CASE eCommand OF
	MC_NoCmd :
		CASE sCurrentState.eStatus OF
			MS_Init :
				IF bEnable THEN
					CASE sCurrentState.eStep OF
						SP_InitStp1 : (* Init all synchros *)
							bBarrelNeedScan := FALSE;
							bArea1StickWarning := FALSE;
							bArea2StickWarning := FALSE;
							bArea3StickWarning := FALSE;
							bArea4StickWarning := FALSE;
							FOR i:=1 TO iMaxSection DO
								FOR j:=1 TO iMaxPosition DO
									abStickPresent[1,i,j]:= FALSE;
									abStickPresent[2,i,j]:= FALSE;
								END_FOR
							END_FOR
							sCurrentState.eStep := SP_InitStp2;
						SP_InitStp2 : (* Lower jacks *)
							bMoveJackUp := FALSE;
							sCurrentState.eStep := SP_InitStp3;
						SP_InitStp3 : (* Check if jacks are down *)
							IF bJackIsDown THEN
								sCurrentState.eStep := SP_InitStp4;
							END_IF
						SP_InitStp4 : (* Lower index *)
							bIndexTable := FALSE;
							sCurrentState.eStep := SP_InitStp5;
						SP_InitStp5 : (* Check if index are down *)
							IF bJackIsDown AND bTableNotIndexed THEN
								sCurrentState.eStep := SP_InitStp6;
							END_IF
						SP_InitStp6 : (* Init barrel axis if modules are safe*)
							eMoveBarrelAxisCommand := AC_Init;
							sCurrentState.eStep := SP_InitStp7;
						SP_InitStp7 : (* Wait init barrel is done*)
							IF TBarrelAxis.eCurrentState = AS_InPosition THEN
								IF bUseNewBarrelFunction THEN
									sCurrentState.eStep := SP_InitStp30;
								ELSE
									sCurrentState.eStep := SP_InitStp10;
								END_IF
							END_IF
						SP_InitStp10 : (* Mono section to use *)
							iIndexPosition := 1;
							IF NOT bSection1IsUsed AND NOT bSection2IsUsed THEN (* no section used *)
								iIndexSection := 1;
								sCurrentState.eStep := SP_InitStp17;
							ELSIF NOT bSection1IsUsed THEN (* section 1 not used *)
								iIndexSection := iStickUsedSection2 + 1;
								iScanPearling:= 2;
								bStickFound := FALSE;
								sCurrentState.eStep := SP_InitStp11;
							ELSE
								iIndexSection := iStickUsedSection1 + 1;
								iScanPearling:= 1;
								bStickFound := FALSE;
								sCurrentState.eStep := SP_InitStp11;
							END_IF
						SP_InitStp11 : (* Turn the barrel to go to the check stick*)
							lrBarrelTargetPos := alrIndexSectionPosition[iIndexSection, iIndexPosition] + lrBarrelCheckPos - alrIndexSectionPosition[1, 1];
							eMoveBarrelAxisCommand := AC_MoveAtAbsPos;
							bStartTimer := FALSE;
							sCurrentState.eStep := SP_InitStp13;
						SP_InitStp13 : (* Wait until position is reached to start the timer *)
							IF (TBarrelAxis.eCurrentState = AS_InPosition) THEN
								bStartTimer := TRUE;
								sCurrentState.eStep := SP_InitStp15;
							END_IF
						SP_InitStp15: (* Wait until the end of timer to detect if the stick is here *)
							IF TBarrelDetectionTimer.Q THEN
								bStartTimer := FALSE;
								abStickPresent[iScanPearling,iIndexSection, iIndexPosition] := bStickPresent;
								IF (bStickPresent) THEN bStickFound := TRUE; END_IF
								iIndexPosition := iIndexPosition + 1;
								IF (iIndexPosition > iMaxPosition) THEN
									CASE iIndexSection OF
										1 :
											bArea1StickWarning := NOT bStickFound;
										2 :
											bArea2StickWarning := NOT bStickFound;
										3 :
											bArea3StickWarning := NOT bStickFound;
										4 :
											bArea4StickWarning := NOT bStickFound;
									END_CASE
									bStickFound := FALSE;
									iIndexPosition := 1;
									iScanPearling:=iScanPearling + 1;
									IF (iScanPearling > 2)  OR (iStickUsedSection1 = iStickUsedSection2) OR NOT bSection2IsUsed THEN
										IF NOT bSection1IsUsed THEN
											iIndexSection := iStickUsedSection2 + 1;
										ELSE
											iIndexSection := iStickUsedSection1 + 1;
										END_IF
										sCurrentState.eStep := SP_InitStp17;
									ELSE
										iIndexSection:= iStickUsedSection2 + 1;
										sCurrentState.eStep := SP_InitStp11;
									END_IF
								ELSE
									sCurrentState.eStep := SP_InitStp11;
								END_IF
							END_IF
						SP_InitStp17 : (* Move to taken,section used 1, 1 *)
							lrBarrelTargetPos := alrIndexSectionPosition[iIndexSection, iIndexPosition] + lrBarrelTakenPos - alrIndexSectionPosition[1, 1];
							eMoveBarrelAxisCommand := AC_MoveAtAbsPos;
							sCurrentState.eStep := SP_InitStp19;
						SP_InitStp19 : (* Wait until position is reached  *)
							IF (TBarrelAxis.eCurrentState = AS_InPosition) THEN
								sCurrentState.eStep := SP_InitStp99;
							END_IF
						SP_InitStp30 : (* Multi section to use *)
							iIndexPosition := 1;
							IF NOT bSection1IsUsed AND NOT bSection2IsUsed THEN (* no section used *)
								iIndexSection := 1;
								sCurrentState.eStep := SP_InitStp37;
							ELSIF NOT bSection1IsUsed THEN (* section 1 not used *)
								yMultiSection2Use := INT_TO_BYTE(iStickUsedSection2);
								iScanPearling:= 2;
								bStickFound := FALSE;
								sCurrentState.eStep := SP_InitStp31;
							ELSE
								yMultiSection2Use := INT_TO_BYTE(iStickUsedSection1);
								iScanPearling:= 1;
								bStickFound := FALSE;
								sCurrentState.eStep := SP_InitStp31;
							END_IF
						SP_InitStp31 :
							iIndexSection := BYTE_TO_INT( yGetActiveSection(yMultiSection2Use));
							IF iIndexSection = 0 THEN
								iIndexSection := 1;
								sCurrentState.eStep := SP_InitStp37;
							ELSE
								sCurrentState.eStep := SP_InitStp32;
							END_IF
						SP_InitStp32 : (* Turn the barrel to go to the check stick*)
							lrBarrelTargetPos := alrIndexSectionPosition[iIndexSection, iIndexPosition] + lrBarrelCheckPos - alrIndexSectionPosition[1, 1];
							eMoveBarrelAxisCommand := AC_MoveAtAbsPos;
							bStartTimer := FALSE;
							sCurrentState.eStep := SP_InitStp33;
						SP_InitStp33 : (* Wait until position is reached to start the timer *)
							IF (TBarrelAxis.eCurrentState = AS_InPosition) THEN
								bStartTimer := TRUE;
								sCurrentState.eStep := SP_InitStp35;
							END_IF
						SP_InitStp35: (* Wait until the end of timer to detect if the stick is here *)
							IF TBarrelDetectionTimer.Q THEN
								bStartTimer := FALSE;
								abStickPresent[iScanPearling,iIndexSection, iIndexPosition] := bStickPresent;
								IF (bStickPresent) THEN bStickFound := TRUE; END_IF
								iIndexPosition := iIndexPosition + 1;
								IF (iIndexPosition > iMaxPosition) THEN
									CASE iIndexSection OF
										1 :
											bArea1StickWarning := NOT bStickFound;
										2 :
											bArea2StickWarning := NOT bStickFound;
										3 :
											bArea3StickWarning := NOT bStickFound;
										4 :
											bArea4StickWarning := NOT bStickFound;
									END_CASE
									bStickFound := FALSE;
									iIndexPosition := 1;
									iIndexSection := BYTE_TO_INT(yGetActiveSection(yMultiSection2Use));
									IF iIndexSection = 0 THEN
										iScanPearling:=iScanPearling + 1;
(*										IF (iScanPearling > 2)  OR (iStickUsedSection1 = iStickUsedSection2) OR NOT bSection2IsUsed THEN*)
										IF (iScanPearling > 2)  OR NOT bSection2IsUsed THEN
											IF NOT bSection1IsUsed THEN
												yMultiSection2Use := INT_TO_BYTE(iStickUsedSection2);
												iIndexSection := BYTE_TO_INT( yGetActiveSection(yMultiSection2Use));
											ELSE
												yMultiSection2Use := INT_TO_BYTE(iStickUsedSection1);
												iIndexSection := BYTE_TO_INT( yGetActiveSection(yMultiSection2Use));
											END_IF
											sCurrentState.eStep := SP_InitStp37;
										ELSE
											yMultiSection2Use := INT_TO_BYTE(iStickUsedSection2);
											sCurrentState.eStep := SP_InitStp31;
										END_IF
									ELSE
										sCurrentState.eStep := SP_InitStp32;
									END_IF
								ELSE
									sCurrentState.eStep := SP_InitStp32;
								END_IF
							END_IF
						SP_InitStp37 : (* Move to taken,section used 1, 1 *)
							lrBarrelTargetPos := alrIndexSectionPosition[iIndexSection, iIndexPosition] + lrBarrelTakenPos - alrIndexSectionPosition[1, 1];
							eMoveBarrelAxisCommand := AC_MoveAtAbsPos;
							sCurrentState.eStep := SP_InitStp39;
						SP_InitStp39 : (* Wait until position is reached  *)
							IF (TBarrelAxis.eCurrentState = AS_InPosition) THEN
								sCurrentState.eStep := SP_InitStp99;
							END_IF
						SP_InitStp99 : (* Leave Init *)
							sCurrentState.eStep := SP_RunStp1;
							sCurrentState.eStatus := MS_Ready;
							sCurrentState.bInitDone := TRUE;
					END_CASE
				ELSE
					sCurrentState.eStatus := MS_Ready;
					sCurrentState.bInitDone := TRUE;
				END_IF
			MS_Running :
				IF bEnable AND  (NOT sCurrentState.bWaitStep) THEN
					CASE sCurrentState.eStep OF
						SP_RunStp1:
							eRunStatus := RS_WaitRequest;
							CASE eRunCommand OF
								RCB_None:
									IF bStopReq  THEN
										sCurrentState.eStatus := MS_Ready;
									ELSIF bPauseReq THEN
										sCurrentState.eStatus := MS_Paused;
									END_IF
								RCB_PrepareStick:
									sCurrentState.eStep := SP_RunStp10;
								RCB_GiveStick:
									sOutStickTake.bHasGiven := FALSE;
									sCurrentState.eStep := SP_RunStp20;
							END_CASE
							IF sCurrentState.eStep<> SP_RunStp1 THEN eRunStatus := RS_ProcessRequest1; END_IF
						SP_RunStp10:(* Prepare Stick *)
							 (* Search Stick *)
							iSearchIndexPosition := 0;
							FOR j:=1 TO 4 DO
								FOR i:=1 TO iMaxPosition DO
									IF abStickPresent[iStickArea,j,i] THEN
										iSearchIndexSection := j;
										iSearchIndexPosition := i;
										EXIT;
									END_IF
								END_FOR
							END_FOR
							IF iSearchIndexPosition = 0 THEN
								bBarrelEmptyError := TRUE;
								sCurrentState.eStep := SP_RunStp1;
							ELSIF iIndexPosition=iSearchIndexPosition AND iIndexSection=iSearchIndexSection AND bTableIndexed THEN
								(* Already prepared *)
								sCurrentState.eStep := SP_RunStp1;
							ELSE
								iIndexPosition := iSearchIndexPosition;
								 iIndexSection := iSearchIndexSection;
								sCurrentState.eStep := SP_RunStp11;
							END_IF
						SP_RunStp11:
							(* Unlock table *)
							bMoveJackUp := FALSE;
							bIndexTable := FALSE;
							sCurrentState.eStep := SP_RunStp12;
						SP_RunStp12: (* Ready to move *)
							IF bJackIsDown AND bTableNotIndexed THEN
								sCurrentState.eStep := SP_RunStp13;
							END_IF
						SP_RunStp13: (* Move to Stick *)
							lrBarrelTargetPos := alrIndexSectionPosition[iIndexSection, iIndexPosition] + lrBarrelTakenPos - alrIndexSectionPosition[1, 1];
							eMoveBarrelAxisCommand := AC_MoveAtAbsPos;
							sCurrentState.eStep := SP_RunStp14;
						SP_RunStp14 : (* Wait until position is reached*)
							IF (TBarrelAxis.eCurrentState = AS_InPosition) THEN
								(* Lock table *)
								bIndexTable := TRUE;
								sCurrentState.eStep := SP_RunStp15;
							END_IF
						SP_RunStp15 :
							IF bTableIndexed THEN
								sCurrentState.eStep := SP_RunStp1;
							END_IF
						SP_RunStp20 : (* Raise the jack when pearling ready*)
							IF NOT bTableIndexed THEN
								bCommandError := TRUE;
							END_IF
							bMoveJackUp := FALSE;
							IF bTableIndexed AND bJackisDown AND sInStickTake.bReadyToTake THEN
								bBarrelNeedScan := TRUE;
								bMoveJackUp := TRUE;
								sCurrentState.eStep := SP_RunStp21;
							END_IF
						SP_RunStp21 : (* Wait for the jack to be up *)
							IF bJackisUp THEN
								sOutStickTake.bHasGiven := TRUE;
								sCurrentState.eStep := SP_RunStp22;
							END_IF
						SP_RunStp22 : (* Wait until the broach has taken the stick *)
							IF sInStickTake.bHasTaken THEN
								sCurrentState.eStep := SP_RunStp23;
							END_IF
						SP_RunStp23 : (* Lower the jack *)
							bMoveJackUp := FALSE;
							sCurrentState.eStep := SP_RunStp24;
						SP_RunStp24 : (* Wait for the jack to go in *)
							IF bJackisDown THEN
								(* Unlock table *)
								bIndexTable := FALSE;
								sCurrentState.eStep := SP_RunStp25;
							END_IF
						SP_RunStp25: (* Check if the stick is still here *)
							IF bTableNotIndexed THEN
								lrBarrelTargetPos := alrIndexSectionPosition[iIndexSection, iIndexPosition] + lrBarrelCheckPos - alrIndexSectionPosition[1, 1];
								eMoveBarrelAxisCommand := AC_MoveAtAbsPos;
								bStartTimer := FALSE;
								sCurrentState.eStep := SP_RunStp26;
							END_IF
						SP_RunStp26 : (* Wait until position is reached to start the timer *)
							IF (TBarrelAxis.eCurrentState = AS_InPosition) THEN
								bStartTimer := TRUE;
								sCurrentState.eStep := SP_RunStp27;
							END_IF
						SP_RunStp27: (* Wait until the end of timer to detect if the stick is still here *)
							IF TBarrelDetectionTimer.Q THEN
								bStartTimer := FALSE;
								abStickPresent[1,iIndexSection, iIndexPosition] := bStickPresent;
								abStickPresent[2,iIndexSection, iIndexPosition] := bStickPresent;
								bBarrelNeedScan := FALSE;
								sOutStickTake.bHasGiven := NOT bStickPresent;
								sCurrentState.eStep := SP_RunStp1;
							END_IF
					END_CASE
				END_IF
			MS_Manual :
				IF NOT bPowerOn THEN
					TManualCmd.TMoveJackUp.Activate := FALSE;
					TManualCmd.TIndexTable.Activate := FALSE;
				END_IF
				TManualCmd.TBarrelAxis.Home.Enable := bJackIsDown AND bTableNotIndexed AND ((TBarrelAxis.eCurrentState = AS_InPosition) OR (TBarrelAxis.eCurrentState = AS_NotHomed)) AND NOT 
bManInterlock;
				TManualCmd.TBarrelAxis.MoveBw.Enable := TBarrelAxis.eCurrentState = AS_InPosition AND bJackIsDown AND bTableNotIndexed AND NOT bManInterlock;
				TManualCmd.TBarrelAxis.MoveFw.Enable := TManualCmd.TBarrelAxis.MoveBw.Enable;
				TManualCmd.TBarrelAxisTakenPos.MoveToTeach.Enable := TManualCmd.TBarrelAxis.MoveBw.Enable;
				TManualCmd.TMoveTaken.TMove1Step.Enable := TManualCmd.TBarrelAxis.MoveBw.Enable;
				TManualCmd.TMoveTaken.TMoveSectionA.Enable := TManualCmd.TBarrelAxis.MoveBw.Enable;
				TManualCmd.TMoveTaken.TMoveSectionB.Enable := TManualCmd.TBarrelAxis.MoveBw.Enable;
				TManualCmd.TMoveTaken.TMoveSectionC.Enable := TManualCmd.TBarrelAxis.MoveBw.Enable;
				TManualCmd.TMoveTaken.TMoveSectionD.Enable := TManualCmd.TBarrelAxis.MoveBw.Enable;
				TManualCmd.TMoveCheck.TMove1Step.Enable := TManualCmd.TBarrelAxis.MoveBw.Enable;
				TManualCmd.TMoveCheck.TMoveSectionA.Enable := TManualCmd.TBarrelAxis.MoveBw.Enable;
				TManualCmd.TMoveCheck.TMoveSectionB.Enable := TManualCmd.TBarrelAxis.MoveBw.Enable;
				TManualCmd.TMoveCheck.TMoveSectionC.Enable := TManualCmd.TBarrelAxis.MoveBw.Enable;
				TManualCmd.TMoveCheck.TMoveSectionD.Enable := TManualCmd.TBarrelAxis.MoveBw.Enable;
				TManualCmd.TBarrelAxisCheckPos.MoveToTeach.Enable := TManualCmd.TBarrelAxis.MoveBw.Enable;
				TManualCmd.TBarrelAxis.CurrentPos := TBarrelAxis.lrCurrentPos;
				TManualCmd.TBarrelAxisTakenPos.TeachedPos := lrBarrelTakenPos;
				TManualCmd.TBarrelAxisCheckPos.TeachedPos := lrBarrelCheckPos;
				TManualCmd.TIndexTable.Enable := ((TBarrelAxis.eCurrentState = AS_InPosition  AND bTableNotIndexed AND TManualCmd.iPosition = 1 AND bJackIsDown) OR bIndexTable) AND bPowerOn;
				TManualCmd.TMoveJackUp.Enable := ((TBarrelAxis.eCurrentState = AS_InPosition AND bTableIndexed AND bJackIsDown) OR bMoveJackUp) AND bPowerOn;
				TManualCmd.iIndexSection := iIndexSection;
				TManualCmd.iIndexPosition := iIndexPosition;
				TManualCmd.bStickPresent := bStickPresent;
				CASE sCurrentState.eStep OF
					SP_ManualStp0 :
						TManualCmd.iPosition := 0; (* 0 undefined, 1 Taken position, 2 Check position , only used for HMI information *)
						TManualCmd.TBarrelAxis.JogStep := lrBarrelJogStep;
						TManualCmd.TBarrelAxis.MoveFw.Activate := FALSE;
						TManualCmd.TBarrelAxis.MoveBw.Activate := FALSE;
						TManualCmd.TBarrelAxisTakenPos.MoveToTeach.Activate := FALSE;
						TManualCmd.TBarrelAxisCheckPos.MoveToTeach.Activate := FALSE;
						TManualCmd.TBarrelAxisTakenPos.Teach := FALSE;
						TManualCmd.TBarrelAxisCheckPos.Teach := FALSE;
						TManualCmd.TMoveJackUp.Activate := bMoveJackUp;
						TManualCmd.TIndexTable.Activate := bIndexTable;
						TManualCmd.TMoveTaken.TMove1Step.Activate := FALSE;
						TManualCmd.TMoveTaken.TMoveSectionA.Activate := FALSE;
						TManualCmd.TMoveTaken.TMoveSectionB.Activate := FALSE;
						TManualCmd.TMoveTaken.TMoveSectionC.Activate := FALSE;
						TManualCmd.TMoveTaken.TMoveSectionD.Activate := FALSE;
						TManualCmd.TMoveCheck.TMove1Step.Activate := FALSE;
						TManualCmd.TMoveCheck.TMoveSectionA.Activate := FALSE;
						TManualCmd.TMoveCheck.TMoveSectionB.Activate := FALSE;
						TManualCmd.TMoveCheck.TMoveSectionC.Activate := FALSE;
						TManualCmd.TMoveCheck.TMoveSectionD.Activate := FALSE;
						TManualCmd.TBarrelAxis.Home.Activate := FALSE;
						sCurrentState.eStep := SP_ManualStp1;
						iIndexSection := iMaxSection;
						iIndexPosition := iMaxPosition;
					SP_ManualStp1:
						IF bStopReq THEN
							sCurrentState.eStatus := MS_Stopped;
						ELSE
							IF (lrBarrelJogStep <> TManualCmd.TBarrelAxis.JogStep) THEN
								lrBarrelJogStep := TManualCmd.TBarrelAxis.JogStep;
							END_IF
							IF TManualCmd.TBarrelAxisTakenPos.Teach THEN
								lrBarrelTakenPos := TBarrelAxis.lrCurrentPos;
								TManualCmd.TBarrelAxisTakenPos.Teach := FALSE;
							END_IF
							IF TManualCmd.TBarrelAxisCheckPos.Teach THEN
								lrBarrelCheckPos := TBarrelAxis.lrCurrentPos;
								TManualCmd.TBarrelAxisCheckPos.Teach := FALSE;
							END_IF
							IF TManualCmd.TBarrelAxisTakenPos.MoveToTeach.Activate THEN
								iIndexPosition := 1;
								iIndexSection := 1;
								lrBarrelTargetPos := TManualCmd.TBarrelAxisTakenPos.TeachedPos;
								sCurrentState.eStep := SP_ManualStp10;
								TManualCmd.iPosition := 1;
							END_IF
							IF TManualCmd.TBarrelAxisCheckPos.MoveToTeach.Activate THEN
								iIndexPosition := 1;
								iIndexSection := 1;
								lrBarrelTargetPos := TManualCmd.TBarrelAxisCheckPos.TeachedPos;
								sCurrentState.eStep := SP_ManualStp10;
								TManualCmd.iPosition := 2;
							END_IF
							IF TManualCmd.TBarrelAxis.MoveBw.Activate THEN
								lrBarrelTargetPos := lrBarrelTargetPos - lrBarrelJogStep;
								sCurrentState.eStep := SP_ManualStp10;
								TManualCmd.iPosition := 0;
							END_IF
							IF TManualCmd.TBarrelAxis.MoveFw.Activate THEN
								lrBarrelTargetPos := lrBarrelTargetPos + lrBarrelJogStep;
								sCurrentState.eStep := SP_ManualStp10;
								TManualCmd.iPosition := 0;
							END_IF
							IF TManualCmd.TMoveTaken.TMove1Step.Activate THEN
								IF (iIndexPosition >= iMaxPosition) THEN
									iIndexPosition := 1;
									IF (iIndexSection >= iMaxSection) THEN
										iIndexSection := 1;
									ELSE
										iIndexSection:= iIndexSection + 1;
									END_IF
								ELSE
									iIndexPosition:= iIndexPosition + 1;
								END_IF
								lrBarrelTargetPos := alrIndexSectionPosition[iIndexSection, iIndexPosition] + lrBarrelTakenPos - alrIndexSectionPosition[1, 1];
								sCurrentState.eStep := SP_ManualStp10;
								TManualCmd.iPosition := 1;
							END_IF
							IF TManualCmd.TMoveTaken.TMoveSectionA.Activate THEN
								iIndexPosition := 1;
								iIndexSection := 1;
								lrBarrelTargetPos := alrIndexSectionPosition[iIndexSection, iIndexPosition] + lrBarrelTakenPos - alrIndexSectionPosition[1, 1];
								sCurrentState.eStep := SP_ManualStp10;
								TManualCmd.iPosition := 1;
							END_IF
							IF TManualCmd.TMoveTaken.TMoveSectionB.Activate THEN
								iIndexPosition := 1;
								iIndexSection := 2;
								lrBarrelTargetPos := alrIndexSectionPosition[iIndexSection, iIndexPosition] + lrBarrelTakenPos - alrIndexSectionPosition[1, 1];
								sCurrentState.eStep := SP_ManualStp10;
								TManualCmd.iPosition := 1;
							END_IF
							IF TManualCmd.TMoveTaken.TMoveSectionC.Activate THEN
								iIndexPosition := 1;
								iIndexSection := 3;
								lrBarrelTargetPos := alrIndexSectionPosition[iIndexSection, iIndexPosition] + lrBarrelTakenPos - alrIndexSectionPosition[1, 1];
								sCurrentState.eStep := SP_ManualStp10;
								TManualCmd.iPosition := 1;
							END_IF
							IF TManualCmd.TMoveTaken.TMoveSectionD.Activate THEN
								iIndexPosition := 1;
								iIndexSection := 4;
								lrBarrelTargetPos := alrIndexSectionPosition[iIndexSection, iIndexPosition] + lrBarrelTakenPos - alrIndexSectionPosition[1, 1];
								sCurrentState.eStep := SP_ManualStp10;
								TManualCmd.iPosition := 1;
							END_IF

							IF TManualCmd.TMoveCheck.TMove1Step.Activate THEN
								IF (iIndexPosition >= iMaxPosition) THEN
									iIndexPosition := 1;
									IF (iIndexSection >= iMaxSection) THEN
										iIndexSection := 1;
									ELSE
										iIndexSection:= iIndexSection + 1;
									END_IF
								ELSE
									iIndexPosition:= iIndexPosition + 1;
								END_IF
								lrBarrelTargetPos := alrIndexSectionPosition[iIndexSection, iIndexPosition] + lrBarrelCheckPos - alrIndexSectionPosition[1, 1];
								sCurrentState.eStep := SP_ManualStp10;
								TManualCmd.iPosition := 2;
							END_IF
							IF TManualCmd.TMoveCheck.TMoveSectionA.Activate THEN
								iIndexPosition := 1;
								iIndexSection := 1;
								lrBarrelTargetPos := alrIndexSectionPosition[iIndexSection, iIndexPosition] + lrBarrelCheckPos - alrIndexSectionPosition[1, 1];
								sCurrentState.eStep := SP_ManualStp10;
								TManualCmd.iPosition := 2;
							END_IF
							IF TManualCmd.TMoveCheck.TMoveSectionB.Activate THEN
								iIndexPosition := 1;
								iIndexSection := 2;
								lrBarrelTargetPos := alrIndexSectionPosition[iIndexSection, iIndexPosition] + lrBarrelCheckPos - alrIndexSectionPosition[1, 1];
								sCurrentState.eStep := SP_ManualStp10;
								TManualCmd.iPosition := 2;
							END_IF
							IF TManualCmd.TMoveCheck.TMoveSectionC.Activate THEN
								iIndexPosition := 1;
								iIndexSection := 3;
								lrBarrelTargetPos := alrIndexSectionPosition[iIndexSection, iIndexPosition] + lrBarrelCheckPos - alrIndexSectionPosition[1, 1];
								sCurrentState.eStep := SP_ManualStp10;
								TManualCmd.iPosition := 2;
							END_IF
							IF TManualCmd.TMoveCheck.TMoveSectionD.Activate THEN
								iIndexPosition := 1;
								iIndexSection := 4;
								lrBarrelTargetPos := alrIndexSectionPosition[iIndexSection, iIndexPosition] + lrBarrelCheckPos - alrIndexSectionPosition[1, 1];
								sCurrentState.eStep := SP_ManualStp10;
								TManualCmd.iPosition := 2;
							END_IF
							IF TManualCmd.TBarrelAxis.Home.Activate AND sCurrentState.eStep = SP_ManualStp1 THEN
								sCurrentState.eStep := SP_ManualStp20;
								TManualCmd.iPosition := 0;
							END_IF
							bMoveJackUp := TManualCmd.TMoveJackUp.Activate;
							bIndexTable := TManualCmd.TIndexTable.Activate;
						END_IF
					SP_ManualStp10: (* Do the movement *)
						eMoveBarrelAxisCommand := AC_MoveModulo;
						sCurrentState.eStep := SP_ManualStp11;
					SP_ManualStp11: (* Wait until position is reached *)
						CASE TBarrelAxis.eCurrentState OF
							AS_InPosition, AS_InError:
								TManualCmd.TBarrelAxisTakenPos.MoveToTeach.Activate := FALSE;
								TManualCmd.TBarrelAxisCheckPos.MoveToTeach.Activate := FALSE;
								TManualCmd.TBarrelAxis.MoveFw.Activate := FALSE;
								TManualCmd.TBarrelAxis.MoveBw.Activate := FALSE;
								TManualCmd.TMoveTaken.TMove1Step.Activate := FALSE;
								TManualCmd.TMoveTaken.TMoveSectionA.Activate := FALSE;
								TManualCmd.TMoveTaken.TMoveSectionB.Activate := FALSE;
								TManualCmd.TMoveTaken.TMoveSectionC.Activate := FALSE;
								TManualCmd.TMoveTaken.TMoveSectionD.Activate := FALSE;
								TManualCmd.TMoveCheck.TMove1Step.Activate := FALSE;
								TManualCmd.TMoveCheck.TMoveSectionA.Activate := FALSE;
								TManualCmd.TMoveCheck.TMoveSectionB.Activate := FALSE;
								TManualCmd.TMoveCheck.TMoveSectionC.Activate := FALSE;
								TManualCmd.TMoveCheck.TMoveSectionD.Activate := FALSE;
								sCurrentState.eStep := SP_ManualStp1;
						END_CASE
					SP_ManualStp20 :  (* Init barrel axis if modules are safe*)
						eMoveBarrelAxisCommand := AC_Home;
						sCurrentState.eStep := SP_ManualStp21;
					SP_ManualStp21 :  (* Turn the barrel to go to init *)
						CASE TBarrelAxis.eCurrentState OF
							AS_InPosition:
								lrBarrelTargetPos := lrBarrelTakenPos;
								eMoveBarrelAxisCommand := AC_MoveAtAbsPos;
								sCurrentState.eStep := SP_ManualStp22;
							AS_InError:
								TManualCmd.TBarrelAxis.Home.Activate := FALSE;
								sCurrentState.eStep := SP_ManualStp1;
						END_CASE
					SP_ManualStp22 :(* Wait until init position is reached *)
						CASE TBarrelAxis.eCurrentState OF
							AS_InPosition, AS_InError:
								sCurrentState.eStep := SP_ManualStp1;
								TManualCmd.TBarrelAxis.Home.Activate := FALSE;
								TManualCmd.iPosition := 1;
								iIndexPosition := 1;
								iIndexSection := 1;
						END_CASE
				END_CASE
			MS_Paused:
				IF bStopReq THEN
					sCurrentState.eStatus := MS_Ready;
				END_IF
		END_CASE;
	MC_Init :
		IF sCurrentState.bInitDone  THEN
			sCurrentState.eStep := SP_InitStp99;
		ELSE
			sCurrentState.eStep := SP_InitStp1;
		END_IF
		sCurrentState.eStatus := MS_Init;
	MC_Run :
		sCurrentState.eStatus := MS_Running;
	MC_Manual :
		sCurrentState.bInitDone := FALSE;
		sCurrentState.eStatus := MS_Manual;
		sCurrentState.eStep := SP_ManualStp0;
	MC_Stop :
		sCurrentState.eStatus := MS_Stopped;
END_CASE;

IF (NOT bPowerOn) THEN
	bMoveJackUp := FALSE;
	bIndexTable := FALSE;
	TManualCmd.TMoveJackUp.Activate := bMoveJackUp;
	TManualCmd.TIndexTable.Activate := bIndexTable;
END_IF

IF bResetErrors THEN
	sCurrentState.bInError := FALSE;
	bCommandError := FALSE;
END_IF

(* Barrel Axis *)
IF (sCurrentState.eStatus = MS_Manual) THEN
	lrCurrentBarrelMoveSpeed := TBarrelAxis.lrManualSpeed;
ELSE
	lrCurrentBarrelMoveSpeed := TBarrelAxis.lrRunningSpeed;
END_IF
TBarrelAxis(
	eCommand		:= eMoveBarrelAxisCommand,
	lrTargetPos		:= lrBarrelTargetPos,
	lrTargetSpeed	:= lrCurrentBarrelMoveSpeed,
	sAxis			:= sBarrelAxisRef,
	bResetErrors		:= bResetErrors,
	bPowerIsOn		:= bPowerOn,
	eHomingAxisType := AHT_OnZeroEncoder,
	stServoButton 	:= TManualCmd.TBarrelAxis.ServoON
);
eMoveBarrelAxisCommand := AC_None;
bBarrelAxisError := (TBarrelAxis.eCurrentState = AS_InError);

(* Check jack error *)
TJack(
	bJackGoOut	:= bMoveJackUp,
	bJackIsIn	:= bJackIsDown,
	bJackIsOut	:= bJackIsUp,
	bResetErrors	:= bResetErrors,
	tTimeOut		:= t#5s,
	bJackError	=> bJackError
);


(* Check table index *)
TTableIndex(
	bJackGoOut	:= bIndexTable,
	bJackIsIn	:= bTableNotIndexed,
	bJackIsOut	:= bTableIndexed,
	bResetErrors	:= bResetErrors,
	bJackError	=> bIndexError
);

IF NOT bEnable THEN
	bModuleError	:= FALSE;
	bBarrelAxisError := FALSE;
	bJackError := FALSE;
	bIndexError := FALSE;
	bArea1StickWarning := FALSE;
	bArea2StickWarning := FALSE;
	bArea3StickWarning := FALSE;
	bArea4StickWarning := FALSE;
END_IF

(* Timer *)
TBarrelDetectionTimer(
	IN	:= bStartTimer,
	PT	:= t#150ms,
	Q	=> ,
	ET	=>
);

sCurrentState.bWarning := bArea1StickWarning OR bArea2StickWarning OR bArea3StickWarning OR bArea4StickWarning;

IF bResetErrors THEN
	bArea1StickWarning := FALSE;
	bArea2StickWarning := FALSE;
	bArea3StickWarning := FALSE;
	bArea4StickWarning := FALSE;
	bBarrelEmptyError := FALSE;
END_IF

IF NOT bPowerOn OR bBarrelAxisError OR bJackError OR bBarrelEmptyError OR bIndexError OR bCommandError THEN
	sCurrentState.bInError := TRUE;
	IF (sCurrentState.eStatus <> MS_Manual) AND (sCurrentState.eStatus <> MS_Stopped) AND (sCurrentState.eStatus <> MS_Init) THEN
		IF bBarrelNeedScan THEN
			sCurrentState.bInitDone := FALSE;
			sCurrentState.eStatus := MS_Stopped;
		ELSE
			sCurrentState.eStatus := MS_Ready;
		END_IF
	END_IF
END_IF

IF NOT bPowerOn OR bBarrelAxisError OR bNewJob THEN
	sCurrentState.bInitDone := FALSE;
	IF (sCurrentState.eStatus <> MS_Manual) THEN
		sCurrentState.eStatus := MS_Stopped;
	END_IF
END_IF

sCurrentState.bInterlocked := bManInterlock AND  (sCurrentState.eStatus = MS_Manual);
bModuleError := sCurrentState.bInError;
sCurrentState.bRunning := (sCurrentState.eStatus = MS_Running);
IF (sCurrentState.eStatus <> MS_Running) THEN eRunStatus := RS_NotRunning; END_IF

END_FUNCTION_BLOCK

// ---- POUs/utils/yGetActiveSection.TcPOU
FUNCTION yGetActiveSection : BYTE
VAR_IN_OUT
	yActiveSections		: BYTE;
END_VAR
VAR
	ySectionChecked		: BYTE;
END_VAR

yGetActiveSection := 0;
WHILE TRUE DO
	ySectionChecked := LREAL_TO_BYTE(EXPT(2,yGetActiveSection));
	yGetActiveSection := yGetActiveSection + 1;
	IF (yActiveSections AND ySectionChecked) > 0 THEN
		(* Section found *)
		yActiveSections := yActiveSections - (yActiveSections AND ySectionChecked);
		EXIT;
	ELSIF yActiveSections = 0 THEN
		yGetActiveSection := 0;
		EXIT;
	END_IF
END_WHILE;

END_FUNCTION

// ---- POUs/Handlers/LiftHdl.TcPOU
FUNCTION_BLOCK LiftHdl

(*
	Description 	: Bloc fonction de gestion du Lift
	Auteur		: DRE
	Date		: 02.09.2016
	Version		: 1.00

	Modifications :

*)

VAR_INPUT
	bEnable						: BOOL;
	bHomeSensor					: BOOL;
	bLimitPos					: BOOL;
	bLimitNeg					: BOOL;
	bDrawerInPos				: BOOL;
	bPlateInPos					: BOOL;
	bPowerOn					: BOOL;
	bResetErrors				: BOOL;
	bStopReq					: BOOL;
	bPauseReq					: BOOL;
	eCommand					: TModuleCommands;
	eLiftType					: TLiftType;
	lrPlateHeight				: LREAL;
	lrPlateEdge					: LREAL;
	lrPlateZOffsetForLift		: LREAL;
	eRunCommand					: TRunCmdLift;
	bNewJob						: BOOL;
	bWaitingForPlates			: BOOL;
	bManInterlock				: BOOL;
	bDrawerLocked				: BOOL;
	bDrawerUnlocked				: BOOL;
	bPlateLocked				: BOOL;
	bPlateUnlocked				: BOOL;
END_VAR
VAR_OUTPUT
	bModuleError				: BOOL;
	bLiftAxisError				: BOOL;
	bLiftEmpty					: BOOL;
	bLiftBlueLight				: BOOL;
	bDrawerIsOpen				: BOOL;
	eRunStatus					: TRunStatus;
	sRunData					: TRunDataLift;
	bNewPlate					: BOOL;
	bLockPlate					: BOOL;
	bUnlockPlate				: BOOL;
	bLockDrawer					: BOOL;
	bUnlockDrawer				: BOOL;
	bLockPlateError				: BOOL;
	bLockDrawerError			: BOOL;
END_VAR
VAR_IN_OUT
	sCurrentState				: TModuleData;
	TManualCmd					: TManLift;
	sLiftAxisRef				: AXIS_REF;
END_VAR
VAR PERSISTENT
	lrLiftEmptyPos				: LREAL					:= 250;		(* Position when Lift is empty *)
	lrLiftFullPos				: LREAL					:= 0;			(* Position when Lift is full *)
	lrLiftLoadPos				: LREAL					:= 10;		(* Position when Drawer can be open *)
	lrLiftJogStep				: LREAL					:= 3;
	lrLiftZOffset				: LREAL					:= 0;
END_VAR
VAR
	eMoveLiftAxisCommand		: TAxisCommands	:= AC_None;
	lrLiftTargetPos				: LREAL;
	lrCurrentLiftMoveSpeed		: LREAL;
	TLiftAxis					: StdAxis;
	bMoveToLoadPlate			: BOOL;
	TCloseTimer					: TON;
	lrLiftPlatePos				: LREAL;
	bLastPowerOn				: BOOL;
	bLastDrawerIsOpen			: BOOL;
	TPlateLocker				: FB_CheckJack1_2;
	TDrawerLocker				: FB_CheckJack1_2;
	bSim4Testing				: BOOL := FALSE;
	bManLockPlate				: BOOL := FALSE;
END_VAR

IF bSim4Testing THEN
	bManInterlock := FALSE;
END_IF

IF (NOT sCurrentState.bStepMode) THEN
	sCurrentState.bWaitStep := FALSE;
END_IF

CASE eCommand OF
	MC_NoCmd :
		CASE sCurrentState.eStatus OF
			MS_Init :
				IF bEnable THEN
				CASE sCurrentState.eStep OF
					SP_InitStp1 :
						bLockDrawer := TRUE;
						bLockPlate := FALSE;
						sCurrentState.eStep := SP_InitStp2;
					SP_InitStp2 :
						IF bDrawerLocked AND bPlateUnlocked THEN
							sCurrentState.eStep := SP_InitStp10;
						END_IF
					SP_InitStp10 :
						(* Init axis*)
						eMoveLiftAxisCommand := AC_Init;
						sCurrentState.eStep := SP_InitStp12;
					SP_InitStp12 : (* Wait init axis is done*)
						IF TLiftAxis.eCurrentState = AS_InPosition THEN
							IF TLiftAxis.lrCurrentPos > lrLiftFullPos THEN
								sCurrentState.eStep := SP_InitStp13;
							ELSE
								sCurrentState.eStep := SP_InitStp20;
							END_IF
						END_IF
					SP_InitStp13: (* we need to go out of the sensor *)
						lrCurrentLiftMoveSpeed := TLiftAxis.lrRunningSpeed;
						//lrLiftTargetPos := TLiftAxis.lrCurrentPos - ( lrLiftZOffset + lrPlateZOffsetForLift + 1);
						lrLiftTargetPos := TLiftAxis.lrCurrentPos - lrPlateZOffsetForLift + lrLiftZOffset;
						IF lrLiftTargetPos < lrLiftFullPos THEN
							lrLiftTargetPos := lrLiftFullPos;
						END_IF
						sCurrentState.eStep := SP_InitStp14;
						eMoveLiftAxisCommand := AC_MoveAtAbsPos;
					SP_InitStp14 : (* Wait out of the plate*)
						IF TLiftAxis.eCurrentState = AS_InPosition THEN
								sCurrentState.eStep := SP_InitStp20;
						END_IF
					SP_InitStp20 :  (* Move to plate*)
						IF  NOT bPlateInPos THEN
							lrLiftTargetPos := lrLiftEmptyPos; (*Go up*)
							sCurrentState.eStep := SP_InitStp21;
						ELSE
							lrLiftTargetPos := lrLiftFullPos; (*Go down*)
							sCurrentState.eStep := SP_InitStp22;
						END_IF
						lrCurrentLiftMoveSpeed := TLiftAxis.stAxisParameters.fRefVeloSearch;
						eMoveLiftAxisCommand := AC_MoveAtAbsPos;
					SP_InitStp21 :  (*moving up, search plate*)
						IF TLiftAxis.eCurrentState = AS_InPosition THEN
							(* Lift is full *)
							sRunData.eLiftPos := LP_Empty;
							sCurrentState.eStep := SP_InitStp99;
						ELSE
							IF  bPlateInPos THEN
								lrLiftTargetPos := lrLiftFullPos; (*Go down*)
								sCurrentState.eStep := SP_InitStp22;
								eMoveLiftAxisCommand := AC_MoveAtAbsPos;
							END_IF
						END_IF
					SP_InitStp22 :(* Moving down, out of sensor*)
						IF TLiftAxis.eCurrentState = AS_InPosition THEN
							 (* Lift is empty *)
							sRunData.eLiftPos := LP_Full;
							sCurrentState.eStep := SP_InitStp99;
						ELSE
							IF  NOT bPlateInPos THEN
								lrCurrentLiftMoveSpeed := TLiftAxis.stAxisParameters.fRefVeloSync;   (* set slow speed*)
								lrLiftTargetPos := lrLiftEmptyPos; (*Go up*)
								sCurrentState.eStep := SP_InitStp23;
								eMoveLiftAxisCommand := AC_MoveAtAbsPos;
							END_IF
						END_IF
					SP_InitStp23 :  (*moving up slowly, search plate*)
						IF TLiftAxis.eCurrentState = AS_InPosition THEN
							(* Lift is full *)
							sRunData.eLiftPos := LP_Empty;
							sCurrentState.eStep := SP_InitStp99;
						ELSE
							IF  bPlateInPos THEN
								lrCurrentLiftMoveSpeed := TLiftAxis.lrRunningSpeed;
								lrLiftPlatePos := TLiftAxis.lrCurrentPos;
								lrLiftTargetPos := lrLiftPlatePos + lrLiftZOffset + lrPlateEdge + lrPlateZOffsetForLift;
								sCurrentState.eStep := SP_InitStp24;
								eMoveLiftAxisCommand := AC_MoveAtAbsPos;
							END_IF
						END_IF
					SP_InitStp24 :(* Wait until position is reached *)
						IF TLiftAxis.eCurrentState = AS_InPosition THEN
							sRunData.eLiftPos := LP_OnPlate;
							IF  bUseLockPlate THEN
								bLockPlate := TRUE;
								sCurrentState.eStep := SP_InitStp25;
							ELSE
								sCurrentState.eStep := SP_InitStp99;
							END_IF
						END_IF
					SP_InitStp25 :
						IF bPlateLocked THEN
							sCurrentState.eStep := SP_InitStp99;
						END_IF
					SP_InitStp99 : (* Leave Init *)
						lrCurrentLiftMoveSpeed := TLiftAxis.lrRunningSpeed;
						sCurrentState.eStep := SP_RunStp1;
						sCurrentState.eStatus := MS_Ready;
						sCurrentState.bInitDone := TRUE;
						bMoveToLoadPlate := FALSE;
						bLiftBlueLight := FALSE;
				END_CASE
				ELSE
					sCurrentState.eStatus := MS_Ready;
					sCurrentState.bInitDone := TRUE;
				END_IF
			MS_Running :
				IF bEnable AND  (NOT sCurrentState.bWaitStep) THEN
					CASE sCurrentState.eStep OF
						SP_RunStp1:
							IF bMoveToLoadPlate THEN
								sCurrentState.eStep := SP_RunStp20;
							ELSE
								eRunStatus := RS_WaitRequest;
								CASE eRunCommand OF
									RCL_None:
										IF bStopReq  THEN
											sCurrentState.eStatus := MS_Ready;
										ELSIF bPauseReq THEN
											sCurrentState.eStatus := MS_Paused;
										END_IF
									RCL_MoveToPlate:
										sRunData.eLiftPos := LP_Moving;
										bLockDrawer := TRUE;
										bLockPlate := FALSE;
										sCurrentState.eStep := SP_RunStp50;
									RCL_MoveToLoadPlate:
										bLockDrawer := TRUE;
										bLockPlate := FALSE;
										sCurrentState.eStep := SP_RunStp20;
									RCL_MoveToOpenDrawer:
										bLockDrawer := TRUE;
										bLockPlate := FALSE;
										sRunData.eLiftPos := LP_Moving;
										sCurrentState.eStep := SP_RunStp30;
								END_CASE
								IF sCurrentState.eStep<> SP_RunStp1 THEN eRunStatus := RS_ProcessRequest1; END_IF
							END_IF
						SP_RunStp20 :  (* Move to load plate*)
							IF bDrawerLocked AND bPlateUnlocked THEN
								bMoveToLoadPlate := FALSE;
								CASE sRunData.eLiftPos OF
									LP_OnPlate:
										IF eLiftType = LT_LOADER THEN
											lrLiftTargetPos := lrLiftPlatePos  + lrLiftZOffset + lrPlateEdge;
										ELSE
											lrLiftTargetPos := lrLiftPlatePos  + lrLiftZOffset + lrPlateEdge - lrPlateHeight ;
										END_IF
										lrCurrentLiftMoveSpeed := TLiftAxis.lrRunningSpeed;
										IF lrLiftTargetPos > TLiftAxis.lrMaxPos THEN
											lrLiftTargetPos := TLiftAxis.lrMaxPos;
										END_IF
										IF lrLiftTargetPos <= lrLiftFullPos THEN
											sRunData.eLiftPos := LP_Full;
											sCurrentState.eStep := SP_RunStp1;
										ELSE
											sRunData.eLiftPos := LP_Moving;
											eMoveLiftAxisCommand := AC_MoveAtAbsPos;
											sCurrentState.eStep := SP_RunStp21;
										END_IF
									LP_OnPlateLoad,LP_Full:
										sCurrentState.eStep := SP_RunStp1;
									LP_Moving, LP_OpenDrawer:
										bMoveToLoadPlate := TRUE;
										sRunData.eLiftPos := LP_Moving;
										sCurrentState.eStep := SP_RunStp50; (* first move to plate *)
									LP_Empty:
										IF eLiftType = LT_LOADER THEN
											sCurrentState.eStep := SP_RunStp1;
										ELSE
											lrLiftTargetPos := lrLiftEmptyPos  + lrLiftZOffset + lrPlateEdge - lrPlateHeight ;
											IF lrLiftTargetPos > TLiftAxis.lrMaxPos THEN
												lrLiftTargetPos := TLiftAxis.lrMaxPos;
											END_IF
											lrCurrentLiftMoveSpeed := TLiftAxis.lrRunningSpeed;
											sRunData.eLiftPos := LP_Moving;
											eMoveLiftAxisCommand := AC_MoveAtAbsPos;
											sCurrentState.eStep := SP_RunStp21;
										END_IF
								END_CASE
							END_IF
						SP_RunStp21 :  (*moving *)
							IF TLiftAxis.eCurrentState = AS_InPosition THEN
								sRunData.eLiftPos := LP_OnPlateLoad;
								sCurrentState.eStep := SP_RunStp1;
							END_IF
						SP_RunStp30 :  (* Move to Open Drawer*)
							IF bDrawerLocked AND bPlateUnlocked THEN
								lrLiftTargetPos := lrLiftLoadPos;
								lrCurrentLiftMoveSpeed := TLiftAxis.lrRunningSpeed;
								eMoveLiftAxisCommand := AC_MoveAtAbsPos;
								sCurrentState.eStep := SP_RunStp31;
							END_IF
						SP_RunStp31 :  (*moving *)
							IF TLiftAxis.eCurrentState = AS_InPosition THEN
								sRunData.eLiftPos := LP_OpenDrawer;
								sCurrentState.eStep := SP_RunStp32;
								bLiftBlueLight := TRUE;
								bLockDrawer := FALSE;
							END_IF
						SP_RunStp32 :  (* Operator open drawer *)
							IF bStopReq  THEN
								sCurrentState.eStatus := MS_Ready;
								sCurrentState.eStep := SP_RunStp33;
							ELSIF bPauseReq THEN
								sCurrentState.eStatus := MS_Paused;
								sCurrentState.eStep := SP_RunStp33;
							END_IF
							IF NOT bDrawerInPos THEN
								TCloseTimer(IN := FALSE);
								sCurrentState.eStep := SP_RunStp33;
							END_IF
						SP_RunStp33 :  (* Operator close drawer *)
							IF bStopReq  THEN
								sCurrentState.eStatus := MS_Ready;
							ELSIF bPauseReq THEN
								sCurrentState.eStatus := MS_Paused;
							END_IF
							TCloseTimer(IN := bDrawerInPos AND NOT bWaitingForPlates, PT := t#3s);
							IF TCloseTimer.Q THEN
								bLockDrawer := TRUE;
								bLiftBlueLight := FALSE;
								sCurrentState.eStep := SP_RunStp1;
							END_IF
						SP_RunStp50 : (* Wait init axis is done*)
							IF bDrawerLocked AND bPlateUnlocked THEN
								IF  sRunData.eLiftPos = LP_OnPlate THEN
									sCurrentState.eStep := SP_RunStp1;
								ELSE
									IF TLiftAxis.eCurrentState = AS_InPosition THEN
										IF TLiftAxis.lrCurrentPos > lrLiftFullPos THEN
											sCurrentState.eStep := SP_RunStp51;
										ELSE
											sCurrentState.eStep := SP_RunStp53;
										END_IF
									END_IF
								END_IF
							END_IF
						SP_RunStp51: (* we need to go out of the sensor *)
							lrCurrentLiftMoveSpeed := TLiftAxis.lrRunningSpeed;
							//lrLiftTargetPos := TLiftAxis.lrCurrentPos - ( lrLiftZOffset + lrPlateZOffsetForLift + 1);
							lrLiftTargetPos := TLiftAxis.lrCurrentPos - lrPlateZOffsetForLift + lrLiftZOffset;
							IF lrLiftTargetPos < lrLiftFullPos THEN
								lrLiftTargetPos := lrLiftFullPos;
							END_IF
							sCurrentState.eStep := SP_RunStp52;
							eMoveLiftAxisCommand := AC_MoveAtAbsPos;
						SP_RunStp52 : (* Wait out of the plate*)
							IF TLiftAxis.eCurrentState = AS_InPosition THEN
									sCurrentState.eStep := SP_RunStp53;
							END_IF
						SP_RunStp53 :  (* Move to plate*)
							IF  NOT bPlateInPos THEN
								lrLiftTargetPos := lrLiftEmptyPos; (*Go up*)
								sCurrentState.eStep := SP_RunStp54;
							ELSE
								lrLiftTargetPos := lrLiftFullPos; (*Go down*)
								sCurrentState.eStep := SP_RunStp55;
							END_IF
							lrCurrentLiftMoveSpeed := TLiftAxis.stAxisParameters.fRefVeloSearch;
							eMoveLiftAxisCommand := AC_MoveAtAbsPos;
						SP_RunStp54 :  (*moving up, search plate*)
							IF TLiftAxis.eCurrentState = AS_InPosition THEN
								(* Lift is full *)
								sRunData.eLiftPos := LP_Empty;
								lrCurrentLiftMoveSpeed := TLiftAxis.lrRunningSpeed;
								sCurrentState.eStep := SP_RunStp1;
							ELSE
								IF  bPlateInPos THEN
									lrLiftTargetPos := lrLiftFullPos; (*Go down*)
									sCurrentState.eStep := SP_RunStp55;
									eMoveLiftAxisCommand := AC_MoveAtAbsPos;
								END_IF
							END_IF
						SP_RunStp55 :(* Moving down, out of sensor*)
							IF TLiftAxis.eCurrentState = AS_InPosition THEN
								 (* Lift is empty *)
								sRunData.eLiftPos := LP_Full;
								lrCurrentLiftMoveSpeed := TLiftAxis.lrRunningSpeed;
								sCurrentState.eStep := SP_RunStp1;
							ELSE
								IF  NOT bPlateInPos THEN
									lrCurrentLiftMoveSpeed := TLiftAxis.stAxisParameters.fRefVeloSync;   (* set slow speed*)
									lrLiftTargetPos := lrLiftEmptyPos; (*Go up*)
									sCurrentState.eStep := SP_RunStp56;
									eMoveLiftAxisCommand := AC_MoveAtAbsPos;
								END_IF
							END_IF
						SP_RunStp56 :  (*moving up slowly, search plate*)
							IF TLiftAxis.eCurrentState = AS_InPosition THEN
								(* Lift is full *)
								sRunData.eLiftPos := LP_Empty;
								lrCurrentLiftMoveSpeed := TLiftAxis.lrRunningSpeed;
								sCurrentState.eStep := SP_RunStp1;
							ELSE
								IF  bPlateInPos THEN
									lrCurrentLiftMoveSpeed := TLiftAxis.lrRunningSpeed;
									lrLiftPlatePos := TLiftAxis.lrCurrentPos;
									lrLiftTargetPos := lrLiftPlatePos + lrPlateEdge + lrLiftZOffset + lrPlateZOffsetForLift;
									sCurrentState.eStep := SP_RunStp57;
									eMoveLiftAxisCommand := AC_MoveAtAbsPos;
								END_IF
							END_IF
						SP_RunStp57 :(* Wait until position is reached *)
							IF TLiftAxis.eCurrentState = AS_InPosition THEN
								(* Lock plate *)
								IF bUseLockPlate THEN
									bLockPlate := TRUE;
								END_IF
								sCurrentState.bWaitStep := TRUE;
								sCurrentState.eStep := SP_RunStp58;
							END_IF
						SP_RunStp58:
							IF bPlateLocked OR NOT bLockPlate THEN
								sRunData.eLiftPos := LP_OnPlate;
								sCurrentState.eStep := SP_RunStp1;
							END_IF
					END_CASE
				END_IF
			MS_Manual :
				TManualCmd.TLiftAxis.Home.Enable := NOT bManInterlock AND bDrawerInPos AND bPlateUnlocked AND ((TLiftAxis.eCurrentState = AS_InPosition) OR (TLiftAxis.eCurrentState = AS_NotHomed));
				TManualCmd.TLiftAxis.MoveBw.Enable := NOT bManInterlock AND bDrawerInPos AND bPlateUnlocked AND (TLiftAxis.eCurrentState = AS_InPosition)  AND (TLiftAxis.lrCurrentPos-lrLiftJogStep >= TLiftAxis.lrMinPos) ;
				TManualCmd.TLiftAxis.MoveFw.Enable := NOT bManInterlock AND bDrawerInPos AND bPlateUnlocked AND (TLiftAxis.eCurrentState = AS_InPosition)  AND (TLiftAxis.lrCurrentPos+lrLiftJogStep <= TLiftAxis.lrMaxPos) ;
				TManualCmd.TLiftAxisFullPos.MoveToTeach.Enable := NOT bManInterlock AND bDrawerInPos AND bPlateUnlocked AND (TLiftAxis.eCurrentState = AS_InPosition)  AND lrLiftFullPos >= TLiftAxis.lrMinPos AND lrLiftFullPos <= TLiftAxis.lrMaxPos;
				TManualCmd.TLiftAxisEmptyPos.MoveToTeach.Enable := NOT bManInterlock AND bDrawerInPos AND bPlateUnlocked AND (TLiftAxis.eCurrentState = AS_InPosition)  AND lrLiftEmptyPos >= TLiftAxis.lrMinPos AND lrLiftEmptyPos <= TLiftAxis.lrMaxPos;
				TManualCmd.TLiftAxisLoadPos.MoveToTeach.Enable := NOT bManInterlock AND bDrawerInPos AND bPlateUnlocked AND (TLiftAxis.eCurrentState = AS_InPosition)  AND lrLiftLoadPos >= TLiftAxis.lrMinPos AND lrLiftLoadPos <= TLiftAxis.lrMaxPos;
				TManualCmd.TLiftAxisZOffset.MoveToTeach.Enable := FALSE;
				TManualCmd.TLiftAxis.CurrentPos := TLiftAxis.lrCurrentPos;
				TManualCmd.TMoveToPlate.Enable := NOT bManInterlock AND bDrawerInPos AND bPlateUnlocked AND (TLiftAxis.eCurrentState = AS_InPosition);
				TManualCmd.TMoveToPlateVision.Enable := NOT bManInterlock AND bDrawerInPos AND bPlateUnlocked AND (TLiftAxis.eCurrentState = AS_InPosition) AND (lrLiftPlatePos<>0);
				TManualCmd.TLiftAxisFullPos.TeachedPos := lrLiftFullPos;
				TManualCmd.TLiftAxisEmptyPos.TeachedPos := lrLiftEmptyPos;
				TManualCmd.TLiftAxisLoadPos.TeachedPos := lrLiftLoadPos;
				TManualCmd.TLiftAxisZOffset.TeachedPos := lrLiftZOffset;
				TManualCmd.bDrawerInPos := bDrawerInPos;
				TManualCmd.bPlateInPos := bPlateInPos;
				TManualCmd.lrPlatePos := lrLiftPlatePos;
				TManualCmd.TLockDrawer.Enable := NOT bDrawerUnlocked OR (NOT bManInterlock AND bDrawerInPos AND (TLiftAxis.eCurrentState = AS_InPosition));
				TManualCmd.TLockPlate.Enable := NOT bPlateUnlocked OR (NOT bManInterlock AND bDrawerInPos AND (TLiftAxis.eCurrentState = AS_InPosition));
				bLiftBlueLight :=  bDrawerUnlocked AND ((TLiftAxis.bAxisHomed) AND ((TLiftAxis.eCurrentState = AS_InPosition)  OR (TLiftAxis.eCurrentState = AS_PowerOff)) AND (TLiftAxis.lrCurrentPos < lrLiftLoadPos + 0.1));
				CASE sCurrentState.eStep OF
					SP_ManualStp0 :
						TManualCmd.TLiftAxis.JogStep := lrLiftJogStep;
						TManualCmd.TLiftAxis.MoveFw.Activate := FALSE;
						TManualCmd.TLiftAxis.MoveBw.Activate := FALSE;
						TManualCmd.TLiftAxis.Home.Activate := FALSE;
						TManualCmd.TMoveToPlate.Activate := FALSE;

						TManualCmd.TLiftAxisFullPos.MoveToTeach.Activate := FALSE;
						TManualCmd.TLiftAxisEmptyPos.MoveToTeach.Activate := FALSE;
						TManualCmd.TLiftAxisLoadPos.MoveToTeach.Activate := FALSE;
						TManualCmd.TLiftAxisZOffset.MoveToTeach.Activate := FALSE;

						TManualCmd.TLiftAxisFullPos.Teach := FALSE;
						TManualCmd.TLiftAxisEmptyPos.Teach := FALSE;
						TManualCmd.TLiftAxisLoadPos.Teach := FALSE;
						TManualCmd.TLiftAxisZOffset.Teach := FALSE;
						lrLiftPlatePos := 0;
						bManLockPlate := FALSE;

						TManualCmd.TLockDrawer.Activate := bLockDrawer;
						TManualCmd.TLockPlate.Activate := bLockPlate;

						sCurrentState.eStep := SP_ManualStp1;
					SP_ManualStp1:
						IF bStopReq THEN
							sCurrentState.eStatus := MS_Stopped;
						ELSE
							IF (lrLiftJogStep <> TManualCmd.TLiftAxis.JogStep) THEN
								lrLiftJogStep := TManualCmd.TLiftAxis.JogStep;
							END_IF
							IF TManualCmd.TLiftAxisZOffset.Teach THEN
								lrLiftZOffset := TLiftAxis.lrCurrentPos - lrLiftPlatePos;
								TManualCmd.TLiftAxisZOffset.Teach := FALSE;
							END_IF
							IF TManualCmd.TLiftAxisFullPos.Teach THEN
								lrLiftFullPos := TLiftAxis.lrCurrentPos;
								TManualCmd.TLiftAxisFullPos.Teach := FALSE;
							END_IF

							IF TManualCmd.TLiftAxisEmptyPos.Teach THEN
								lrLiftEmptyPos := TLiftAxis.lrCurrentPos;
								TManualCmd.TLiftAxisEmptyPos.Teach := FALSE;
							END_IF
							IF TManualCmd.TLiftAxisLoadPos.Teach THEN
								lrLiftLoadPos := TLiftAxis.lrCurrentPos;
								TManualCmd.TLiftAxisLoadPos.Teach := FALSE;
							END_IF
							IF TManualCmd.TLiftAxisFullPos.MoveToTeach.Activate THEN
								lrLiftTargetPos := TManualCmd.TLiftAxisFullPos.TeachedPos;
								sCurrentState.eStep := SP_ManualStp10;
							END_IF

							IF TManualCmd.TLiftAxisEmptyPos.MoveToTeach.Activate THEN
								lrLiftTargetPos := TManualCmd.TLiftAxisEmptyPos.TeachedPos;
								sCurrentState.eStep := SP_ManualStp10;
							END_IF
							IF TManualCmd.TLiftAxisLoadPos.MoveToTeach.Activate THEN
								lrLiftTargetPos := TManualCmd.TLiftAxisLoadPos.TeachedPos;
								sCurrentState.eStep := SP_ManualStp10;
							END_IF
							IF TManualCmd.TLiftAxis.MoveBw.Activate THEN
								lrLiftTargetPos := lrLiftTargetPos - lrLiftJogStep;
								sCurrentState.eStep := SP_ManualStp10;
							END_IF
							IF TManualCmd.TLiftAxis.MoveFw.Activate THEN
								lrLiftTargetPos := lrLiftTargetPos + lrLiftJogStep;
								sCurrentState.eStep := SP_ManualStp10;
							END_IF
							IF TManualCmd.TMoveToPlate.Activate THEN
								TManualCmd.TMoveToPlate.Activate := FALSE;
								sCurrentState.eStep := SP_ManualStp30;
							END_IF
							IF TManualCmd.TMoveToPlateVision.Activate THEN
								TManualCmd.TMoveToPlateVision.Activate := FALSE;
								lrLiftTargetPos := lrLiftPlatePos + lrLiftZOffset + lrPlateZOffsetForLift;
								sCurrentState.eStep := SP_ManualStp10;
							END_IF
							IF TManualCmd.TLiftAxis.Home.Activate AND sCurrentState.eStep = SP_ManualStp1 THEN
								sCurrentState.eStep := SP_ManualStp20;
							END_IF
							IF sCurrentState.eStep <> SP_ManualStp1 THEN
								bManLockPlate := FALSE;
							END_IF
						END_IF
					SP_ManualStp10: (* Do the movement *)
						eMoveLiftAxisCommand := AC_MoveAtAbsPos;
						lrCurrentLiftMoveSpeed := TLiftAxis.lrManualSpeed;
						sCurrentState.eStep := SP_ManualStp11;
					SP_ManualStp11: (* Wait until position is reached *)
						CASE TLiftAxis.eCurrentState OF
							AS_InPosition, AS_InError:
								TManualCmd.TLiftAxis.MoveFw.Activate := FALSE;
								TManualCmd.TLiftAxis.MoveBw.Activate := FALSE;
								TManualCmd.TLiftAxis.Home.Activate := FALSE;
		
								TManualCmd.TLiftAxisFullPos.MoveToTeach.Activate := FALSE;
								TManualCmd.TLiftAxisEmptyPos.MoveToTeach.Activate := FALSE;
								TManualCmd.TLiftAxisLoadPos.MoveToTeach.Activate := FALSE;
								sCurrentState.eStep := SP_ManualStp1;
						END_CASE
					SP_ManualStp20 :  (* Homing lift axis if modules are safe*)
						eMoveLiftAxisCommand := AC_Home;
						sCurrentState.eStep := SP_ManualStp21;
					SP_ManualStp21 :  (* Move lift to go to load *)
						CASE TLiftAxis.eCurrentState OF
							AS_InPosition:
								lrCurrentLiftMoveSpeed := TLiftAxis.lrManualSpeed;
								lrLiftTargetPos := lrLiftLoadPos;
								eMoveLiftAxisCommand := AC_MoveAtAbsPos;
								sCurrentState.eStep := SP_ManualStp22;
							AS_InError:
								TManualCmd.TLiftAxis.Home.Activate := FALSE;
								sCurrentState.eStep := SP_ManualStp1;
						END_CASE
					SP_ManualStp22 :(* Wait until init position is reached *)
						CASE TLiftAxis.eCurrentState OF
							AS_InPosition, AS_InError:
								sCurrentState.eStep := SP_ManualStp1;
								TManualCmd.TLiftAxis.Home.Activate := FALSE;
						END_CASE
					SP_ManualStp30 :  (* Move to plate*)
						IF  NOT bPlateInPos THEN
							lrLiftTargetPos := lrLiftEmptyPos; (*Go up*)
							sCurrentState.eStep := SP_ManualStp31;
						ELSE
							lrLiftTargetPos := lrLiftFullPos; (*Go down*)
							sCurrentState.eStep := SP_ManualStp32;
						END_IF
						lrCurrentLiftMoveSpeed := TLiftAxis.stAxisParameters.fRefVeloSearch;
						eMoveLiftAxisCommand := AC_MoveAtAbsPos;
					SP_ManualStp31 :  (*moving up, search plate*)
						CASE TLiftAxis.eCurrentState OF
							AS_InPosition: (* Lift is full *)
								sCurrentState.eStep := SP_ManualStp1;
							AS_InError:
								sCurrentState.eStep := SP_ManualStp1;
							ELSE
								IF  bPlateInPos THEN
									lrLiftTargetPos := lrLiftFullPos; (*Go down*)
									sCurrentState.eStep := SP_ManualStp32;
									eMoveLiftAxisCommand := AC_MoveAtAbsPos;
								END_IF
						END_CASE
					SP_ManualStp32 :(* Moving down, out of sensor*)
						CASE TLiftAxis.eCurrentState OF
							AS_InPosition: (* Lift is empty *)
								sCurrentState.eStep := SP_ManualStp1;
							AS_InError:
								sCurrentState.eStep := SP_ManualStp1;
							ELSE
								IF  NOT bPlateInPos THEN
									lrCurrentLiftMoveSpeed := TLiftAxis.stAxisParameters.fRefVeloSync;   (* set slow speed*)
									lrLiftTargetPos := lrLiftEmptyPos; (*Go up*)
									sCurrentState.eStep := SP_ManualStp33;
									eMoveLiftAxisCommand := AC_MoveAtAbsPos;
								END_IF
						END_CASE
					SP_ManualStp33 :  (*moving up slowly, search plate*)
						CASE TLiftAxis.eCurrentState OF
							AS_InPosition: (* Lift is full *)
								sCurrentState.eStep := SP_ManualStp1;
							AS_InError:
								sCurrentState.eStep := SP_ManualStp1;
							ELSE
								IF  bPlateInPos THEN
									lrCurrentLiftMoveSpeed := TLiftAxis.lrManualSpeed;
									lrLiftPlatePos := TLiftAxis.lrCurrentPos;
									lrLiftTargetPos := lrLiftPlatePos; (*Move to current pos*)
									sCurrentState.eStep := SP_ManualStp34;
									eMoveLiftAxisCommand := AC_MoveAtAbsPos;
								END_IF
						END_CASE
					SP_ManualStp34 :(* Wait until position is reached *)
						CASE TLiftAxis.eCurrentState OF
							AS_InPosition:
								bManLockPlate := TRUE;
								sCurrentState.eStep := SP_ManualStp1;
							AS_InError:
								sCurrentState.eStep := SP_ManualStp1;
						END_CASE
				END_CASE
				bLockDrawer := TManualCmd.TLockDrawer.Activate;
				bLockPlate := TManualCmd.TLockPlate.Activate;
			MS_Paused:
				IF bStopReq THEN
					sCurrentState.eStatus := MS_Ready;
				END_IF
		END_CASE;
	MC_Init :
		IF sCurrentState.bInitDone THEN
			sCurrentState.eStep := SP_InitStp99;
		ELSE
			sCurrentState.eStep := SP_InitStp1;
		END_IF
		sCurrentState.eStatus := MS_Init;
	MC_Run :
		sCurrentState.eStatus := MS_Running;
	MC_Manual :
		sCurrentState.bInitDone := FALSE;
		sCurrentState.eStatus := MS_Manual;
		sCurrentState.eStep := SP_ManualStp0;
	MC_Stop :
		sCurrentState.eStatus := MS_Stopped;
		eMoveLiftAxisCommand := AC_Stop;
END_CASE;

IF bResetErrors THEN
	sCurrentState.bInError := FALSE;
END_IF

IF NOT bDrawerInPos AND (TLiftAxis.eCurrentState = AS_Moving OR TLiftAxis.eCurrentState = AS_Homing) THEN
	eMoveLiftAxisCommand := AC_ForceStop;
END_IF

(* Barrel Axis *)
IF (sCurrentState.eStatus = MS_Manual) AND (	lrCurrentLiftMoveSpeed > TLiftAxis.lrManualSpeed) THEN
	lrCurrentLiftMoveSpeed := TLiftAxis.lrManualSpeed;
END_IF
TLiftAxis(
	eCommand		:= eMoveLiftAxisCommand,
	lrTargetPos		:= lrLiftTargetPos,
	lrTargetSpeed	:= lrCurrentLiftMoveSpeed,
	sAxis			:= sLiftAxisRef,
	bResetErrors	:= bResetErrors,
	bHomeSensor		:= bHomeSensor,
	bPowerIsOn		:= bPowerOn,
	bPosLimitSwitch	:= NOT bLimitPos,
	bNegLimitSwitch	:= NOT bLimitNeg,
	lrMoveOutDist	:= 10,
	stServoButton 	:= TManualCmd.TLiftAxis.ServoON
);
eMoveLiftAxisCommand := AC_None;
bLiftAxisError := (TLiftAxis.eCurrentState = AS_InError);

(* Check Plate locker Error *)
TPlateLocker(
	bJackGoOut		:= bLockPlate,
	bJackIsIn		:= bPlateUnlocked,
	bJackIsOut		:= bPlateLocked,
	tTimeOut		:= T#1S,
	bResetErrors	:= bResetErrors,
	bJackError		=> bLockPlateError
);
bUnlockPlate := NOT bLockPlate;

(* Check Drawer locker Error *)
TDrawerLocker(
	bJackGoOut		:= bLockDrawer,
	bJackIsIn		:= bDrawerUnlocked,
	bJackIsOut		:= bDrawerLocked,
	tTimeOut		:= T#1S,
	bResetErrors	:= bResetErrors,
	bJackError		=> bLockDrawerError
);
bUnlockDrawer := NOT bLockDrawer;

IF NOT bEnable THEN
	bModuleError	:= FALSE;
	bLiftAxisError := FALSE;
	bLockDrawerError := FALSE;
	bLockPlateError := FALSE;
END_IF
bDrawerIsOpen := NOT bDrawerInPos;
sCurrentState.bWarning := bDrawerIsOpen OR bLiftBlueLight OR bWaitingForPlates;

IF bResetErrors THEN
	bLiftEmpty := FALSE;
END_IF

IF NOT bPowerOn OR bLiftAxisError OR bLockDrawerError OR bLockPlateError THEN
	sCurrentState.bInError := TRUE;
	IF (sCurrentState.eStatus <> MS_Manual) AND (sCurrentState.eStatus <> MS_Stopped) AND (sCurrentState.eStatus <> MS_Init) THEN
		sCurrentState.eStatus := MS_Ready;
	END_IF
END_IF

IF NOT bPowerOn OR bLiftAxisError OR bNewJob OR bLockDrawerError OR bLockPlateError THEN
	sCurrentState.bInitDone := FALSE;
	IF (sCurrentState.eStatus <> MS_Manual) THEN
		sCurrentState.eStatus := MS_Stopped;
	END_IF
END_IF

bNewPlate := FALSE;
IF bPowerOn <> bLastPowerOn THEN
	bLastPowerOn := bPowerOn;
	IF NOT bPowerOn THEN
		bNewPlate := bNewPlate; (* Dummy instruction, can be removed *)
		(*bNewPlate := TRUE;*)
	END_IF
END_IF
IF bDrawerIsOpen <> bLastDrawerIsOpen THEN
	bLastDrawerIsOpen := bDrawerIsOpen;
	IF bDrawerIsOpen THEN
		bNewPlate := TRUE;
	END_IF
END_IF

sCurrentState.bInterlocked := bManInterlock AND  (sCurrentState.eStatus = MS_Manual);
bModuleError := sCurrentState.bInError;
sCurrentState.bRunning := (sCurrentState.eStatus = MS_Running);
IF (sCurrentState.eStatus <> MS_Running) THEN eRunStatus := RS_NotRunning; END_IF

END_FUNCTION_BLOCK

// ---- POUs/Handlers/RejectHdl.TcPOU
FUNCTION_BLOCK RejectHdl
(*
	Description 	: Bloc fonction de gestion du rejet
	Auteur		: DRE
	Date		: 06.09.2016
	Version		: 1.00

	Modifications :

*)

VAR_INPUT
	bEnable						: BOOL;
	bDrawerInPos				: BOOL;
	bPlateInPos					: BOOL;
	bPowerOn					: BOOL;
	bResetErrors					: BOOL;
	bStopReq					: BOOL;
	bPauseReq					: BOOL;
	eCommand					: TModuleCommands;
	eRunCommand				: TRunCmdReject;
	bWaitingForPlates				: BOOL;
END_VAR
VAR_OUTPUT
	bModuleError					: BOOL;
	bDrawerIsOpen				: BOOL;
	bDrawerOpenedError			: BOOL;
	bNoPlatePresent				: BOOL;
	bRejectBlueLight				: BOOL;
	eRunStatus					: TRunStatus;
	sRunData					: TRunDataReject;
	bNewPlate					: BOOL;
END_VAR
VAR_IN_OUT
	sCurrentState					: TModuleData;
	TManualCmd					: TManReject;
END_VAR
VAR
	TCloseTimer					: TON;
	bPlateReady					: BOOL;
	bLastPlateReady				: BOOL;
END_VAR
VAR PERSISTENT
	RejectPlateNb				:DWORD;
END_VAR

IF (NOT sCurrentState.bStepMode) THEN
	sCurrentState.bWaitStep := FALSE;
END_IF

CASE eCommand OF
	MC_NoCmd :
		CASE sCurrentState.eStatus OF
			MS_Init :
				IF bEnable THEN
				CASE sCurrentState.eStep OF
					SP_InitStp1 : (* Init all synchros *)
						bRejectBlueLight := TRUE;
						sCurrentState.eStep := SP_InitStp99;
					SP_InitStp99 : (* Leave Init *)
						sCurrentState.eStep := SP_RunStp1;
						sCurrentState.eStatus := MS_Ready;
						sCurrentState.bInitDone := TRUE;
				END_CASE
				ELSE
					sCurrentState.eStatus := MS_Ready;
					sCurrentState.bInitDone := TRUE;
				END_IF
			MS_Running :
				IF bEnable AND  (NOT sCurrentState.bWaitStep) THEN
					CASE sCurrentState.eStep OF
						SP_RunStp1 :(* Wait request *)
							eRunStatus := RS_WaitRequest;
							CASE eRunCommand OF
								RCR_None:
									IF bStopReq  THEN
										sCurrentState.eStatus := MS_Ready;
									ELSIF bPauseReq  THEN
										sCurrentState.eStatus := MS_Paused;
									ELSIF NOT bDrawerInPos OR NOT bPlateInPos THEN
										sCurrentState.eStep := SP_RunStp10;
									END_IF
								RCR_OpenDrawer:
									sCurrentState.eStep := SP_RunStp10;
								RCR_LockDrawer:
									IF bDrawerInPos AND bPlateInPos THEN
										bRejectBlueLight := FALSE;
									END_IF
									sCurrentState.eStep := SP_RunStp1;
								RCR_UnlockDrawer:
									bRejectBlueLight := TRUE;
									sCurrentState.eStep := SP_RunStp1;
							END_CASE
							IF sCurrentState.eStep<> SP_RunStp1 THEN
								IF NOT bRejectBlueLight THEN
									bDrawerOpenedError := TRUE;
								END_IF
								sRunData.eRejectStatus := RS_OpenDrawer;
								eRunStatus := RS_ProcessRequest1;
							ELSE
								IF NOT bRejectBlueLight AND bDrawerInPos AND bPlateInPos THEN
									sRunData.eRejectStatus := RS_Locked;
								ELSIF bDrawerInPos AND bPlateInPos THEN
									sRunData.eRejectStatus := RS_Ready;
								ELSE
									sRunData.eRejectStatus := RS_Empty;
								END_IF
							END_IF
						SP_RunStp10 :  (* Operator open drawer *)
							IF bStopReq  THEN
								sCurrentState.eStatus := MS_Ready;
							ELSIF bPauseReq THEN
								sCurrentState.eStatus := MS_Paused;
							END_IF
							bRejectBlueLight := TRUE;
							IF bDrawerInPos AND bPlateInPos THEN
								TCloseTimer(IN := FALSE);
								sCurrentState.eStep := SP_RunStp11;
							END_IF
;						SP_RunStp11 :  (* Operator close drawer *)
							IF bStopReq  THEN
								sCurrentState.eStatus := MS_Ready;
							ELSIF bPauseReq THEN
								sCurrentState.eStatus := MS_Paused;
							END_IF
							TCloseTimer(IN := bDrawerInPos AND NOT bWaitingForPlates, PT := t#2s);
							IF TCloseTimer.Q THEN
								sCurrentState.eStep := SP_RunStp1;
							END_IF
					END_CASE
				END_IF
			MS_Manual :
				TManualCmd.bDrawerInPos := bDrawerInPos;
				TManualCmd.bPlateInPos := bPlateInPos;
				bRejectBlueLight :=  TRUE;
				IF bStopReq THEN
					sCurrentState.eStatus := MS_Stopped;
				END_IF
			MS_Paused:
				IF bStopReq THEN
					sCurrentState.eStatus := MS_Ready;
				END_IF
			MS_Stopped:
				bRejectBlueLight :=  TRUE;
		END_CASE;
	MC_Init :
		IF sCurrentState.bInitDone THEN
			sCurrentState.eStep := SP_InitStp99;
		ELSE
			sCurrentState.eStep := SP_InitStp1;
		END_IF
		sCurrentState.eStatus := MS_Init;
	MC_Run :
		sCurrentState.eStatus := MS_Running;
	MC_Manual :
		sCurrentState.bInitDone := FALSE;
		sCurrentState.eStatus := MS_Manual;
		sCurrentState.eStep := SP_ManualStp0;
	MC_Stop :
		sCurrentState.eStatus := MS_Stopped;
END_CASE;

bNoPlatePresent := NOT bPlateInPos;

IF bResetErrors THEN
	bDrawerOpenedError := FALSE;
	bNoPlatePresent := FALSE;
	sCurrentState.bInError := FALSE;
END_IF

IF NOT bEnable THEN
	bModuleError	:= FALSE;
END_IF

bNewPlate := FALSE;
bPlateReady := bDrawerInPos AND bPlateInPos;
IF bPlateReady <> bLastPlateReady THEN
	bLastPlateReady := bPlateReady;
	IF NOT bPlateReady THEN
		bNewPlate := TRUE;
		RejectPlateNb := RejectPlateNb + 1;
	END_IF
END_IF
bDrawerIsOpen := NOT bDrawerInPos;
sCurrentState.bWarning := bDrawerIsOpen OR bNoPlatePresent OR bRejectBlueLight OR bWaitingForPlates;

(*
IF bResetErrors THEN
	Nothing to do
END_IF
*)
IF bDrawerOpenedError THEN
	sCurrentState.bInError := TRUE;
	IF (sCurrentState.eStatus <> MS_Manual) AND (sCurrentState.eStatus <> MS_Stopped) AND (sCurrentState.eStatus <> MS_Init) THEN
		sCurrentState.eStatus := MS_Ready;
	END_IF
END_IF

bModuleError := sCurrentState.bInError;

sCurrentState.bRunning := (sCurrentState.eStatus = MS_Running);
IF (sCurrentState.eStatus <> MS_Running) THEN
	sRunData.eRejectStatus := RS_OpenDrawer;
	eRunStatus := RS_NotRunning;
END_IF

END_FUNCTION_BLOCK

// ---- POUs/Handlers/VisionHdl.TcPOU
FUNCTION_BLOCK VisionHdl
(*
	Description 	: Bloc fonction de gestion de la vision
	Auteur		: DRE
	Date		: 07.09.2016
	Version		: 1.00

	Modifications :

*)

VAR_INPUT
	bEnable						: BOOL;
	bNewJob					: BOOL;
	bPowerOn					: BOOL;
	bResetErrors					: BOOL;
	bStopReq					: BOOL;
	bPauseReq					: BOOL;
	bJobInProgress				: BOOL;
	eCommand					: TModuleCommands;
	acVisionRecipeName			: STRING(20);
	eRunCommand				:TRunCmdVision;
END_VAR
VAR_OUTPUT
	bModuleError					: BOOL;
	bNotReady					: BOOL;
	bNotConnected				: BOOL;
	bInSimulation					: BOOL;
	eRunStatus					: TRunStatus;
END_VAR
VAR_IN_OUT
	sCurrentState					: TModuleData;
	TManualCmd					: TManVision;
	TVision						: TVisionData;
	sRunData					: TRunDataVision;
END_VAR
VAR PERSISTENT
	bSimVision					: BOOL;
END_VAR
VAR
	fbNtGetTime					: NT_GetTime;
	bNtGetTime					: BOOL;
(*	bVisionBusy					: BOOL;*)
	eVisionStep					: TModuleSteps := SP_RunStp0;
	eVisionCommand				: TVisionRequest;
	TAliveCheckTimer			: TON;
	bAliveCheck					: BOOL;
	bLastVisionConnected			: BOOL;
	TNow						: TIMESTRUCT;
END_VAR

IF (NOT sCurrentState.bStepMode) THEN
	sCurrentState.bWaitStep := FALSE;
END_IF

CASE eCommand OF
	MC_NoCmd :
		CASE sCurrentState.eStatus OF
			MS_Init :
				IF bEnable THEN
				CASE sCurrentState.eStep OF
					SP_InitStp1 : (* Init all synchros *)
						bNotReady := FALSE;
						IF (TVision.bRequestDone) THEN (* Wait until last command is completed*)
							sCurrentState.eStep := SP_InitStp2;
						END_IF
					SP_InitStp2:
						TVision.acRefFileName := acVisionRecipeName;
						eVisionCommand := VR_Init;
						sCurrentState.eStep := SP_InitStp3;
					SP_InitStp3:
						IF (TVision.bRequestDone) AND (TVision.bReady OR TVision.bConfigMode) THEN
							sCurrentState.eStep := SP_InitStp99;
						ELSIF (TVision.bRequestError) THEN
							bNotReady := TRUE;
						END_IF
					SP_InitStp99 : (* Leave Init *)
						sCurrentState.eStep := SP_RunStp1;
						sCurrentState.eStatus := MS_Ready;
						sCurrentState.bInitDone := TRUE;
				END_CASE
				ELSE
					sCurrentState.eStatus := MS_Ready;
					sCurrentState.bInitDone := TRUE;
				END_IF
			MS_Running :
				IF bEnable AND  (NOT sCurrentState.bWaitStep) THEN
					CASE sCurrentState.eStep OF
						SP_RunStp1:
							eRunStatus := RS_WaitRequest;
							CASE eRunCommand OF
								RCV_None:
									IF bStopReq  THEN
										sCurrentState.eStatus := MS_Ready;
									ELSIF bPauseReq THEN
										sCurrentState.eStatus := MS_Paused;
									END_IF
								RCV_GrabImage:
									sCurrentState.eStep := SP_RunStp10;
								RCV_AnalyseImage:
									sCurrentState.eStep := SP_RunStp20;
							END_CASE
							IF sCurrentState.eStep<> SP_RunStp1 THEN eRunStatus := RS_ProcessRequest1; END_IF
						SP_RunStp10:
							eVisionCommand := VR_GrabImage;
							sCurrentState.eStep := SP_RunStp11;
						SP_RunStp11:
							IF (TVision.bRequestDone) THEN
								sCurrentState.eStep := SP_RunStp1;
							ELSIF (TVision.bRequestError) THEN
								bNotReady := TRUE;
							END_IF
						SP_RunStp20:
							eVisionCommand := VR_Analyse;
							TVision.iUseModel := sRunData.iUseModel;
							sCurrentState.eStep := SP_RunStp21;
						SP_RunStp21:
							IF (TVision.bRequestDone) AND (TVision.bReady) THEN
								sRunData.TVisionPartData := TVision.TPartData;
								sCurrentState.eStep := SP_RunStp1;
							ELSIF (TVision.bRequestError) THEN
								bNotReady := TRUE;
							END_IF

					END_CASE
				END_IF
			MS_Manual :
				TManualCmd.TInit.Enable := TVision.bConnected;
				TManualCmd.TAnalyse.Enable := TVision.bReady;
				TManualCmd.TRun.Enable := TVision.bReady;
				TManualCmd.bConnected := TVision.bConnected;
				TManualCmd.iMaxModel := TVision.iMaxModel;
				TManualCmd.bReady := TVision.bReady;
				TManualCmd.bSimRecipe := TVision.bSimRecipe;
				TManualCmd.TPartData := TVision.TPartData;
				IF NOT TVision.bConnected OR NOT TVision.bReady THEN
					TManualCmd.bPartDataValid := FALSE;
				END_IF
				CASE sCurrentState.eStep OF
					SP_ManualStp0:
						TManualCmd.TInit.Activate := FALSE;
						TManualCmd.TAnalyse.Activate := FALSE;
						TManualCmd.TRun.Activate := FALSE;
						TManualCmd.acVisionRecipeName := TVision.acRefFileName;
						TManualCmd.iUseModel := TVision.iUseModel;
						TManualCmd.bConfigMode.Enable := TRUE;
						TManualCmd.bConfigMode.Activate := TVision.bConfigMode;;
						IF (TVision.bRequestDone) THEN (* Wait until last command is completed*)
							sCurrentState.eStep := SP_ManualStp1;
						END_IF
					SP_ManualStp1:
						IF bStopReq THEN
							sCurrentState.eStatus := MS_Stopped;
						END_IF
						IF TManualCmd.TInit.Activate THEN
							TManualCmd.bPartDataValid := FALSE;
							TManualCmd.TRun.Activate := FALSE;
							TManualCmd.TInit.Activate := FALSE;
							TVision.acRefFileName := TManualCmd.acVisionRecipeName;
							TVision.iMaxModel := 0;
							TVision.iUseModel := 0;
							eVisionCommand := VR_Init;
							TManualCmd.TInitTime := TNow;
							sCurrentState.eStep := SP_ManualStp2;
						END_IF
						IF TManualCmd.TAnalyse.Activate THEN
							TManualCmd.bPartDataValid := FALSE;
							TManualCmd.TRun.Activate := FALSE;
							TManualCmd.TAnalyse.Activate := FALSE;
							eVisionCommand := VR_GrabImage;
							TVision.iUseModel := TManualCmd.iUseModel;
							TManualCmd.TAnalyseTime := TNow;
							sCurrentState.eStep := SP_ManualStp3;
						END_IF
						IF TManualCmd.TRun.Activate THEN
							IF NOT TManualCmd.TRun.Enable THEN
								TManualCmd.TRun.Activate := FALSE;
							ELSE
								eVisionCommand := VR_GrabImage;
								TVision.iUseModel := TManualCmd.iUseModel;
								sCurrentState.eStep := SP_ManualStp3;
							END_IF
						END_IF
						TVision.bConfigMode := TManualCmd.bConfigMode.Activate;
					SP_ManualStp2:
						TManualCmd.bReady := FALSE;
						IF (TVision.bRequestDone) THEN (* Wait until last command is completed*)
							sCurrentState.eStep := SP_ManualStp1;
						END_IF
					SP_ManualStp3: (* Wait for image grabbed *)
						IF (TVision.bRequestDone) THEN
							eVisionCommand := VR_Analyse;
							sCurrentState.eStep := SP_ManualStp4;
						END_IF
					SP_ManualStp4: (* Wait analyse done *)
						IF (TVision.bRequestDone) THEN (* Wait until last command is completed*)
							TManualCmd.bPartDataValid := TRUE;
							sCurrentState.eStep := SP_ManualStp1;
						END_IF
				END_CASE
			MS_Paused:
				IF bStopReq THEN
					sCurrentState.eStatus := MS_Ready;
				END_IF
		END_CASE;
	MC_Init :
		IF sCurrentState.bInitDone THEN
			sCurrentState.eStep := SP_InitStp99;
		ELSE
			sCurrentState.eStep := SP_InitStp1;
		END_IF
		sCurrentState.eStatus := MS_Init;
	MC_Run :
		IF TVision.bConfigMode THEN
			bNotReady := TRUE;
		ELSE
			sCurrentState.eStatus := MS_Running;
		END_IF
	MC_Manual :
		sCurrentState.bInitDone := FALSE;
		sCurrentState.eStatus := MS_Manual;
		sCurrentState.eStep := SP_ManualStp0;
	MC_Stop :
		sCurrentState.eStatus := MS_Stopped;
END_CASE;

(* Vision Com *)
IF (bLastVisionConnected <> TVision.bConnected) THEN
	IF (TVision.bConnected) THEN (*Vision just connected, reset alive and alive timer *)
		bAliveCheck := FALSE;
		TVision.bAlive := FALSE;
		TAliveCheckTimer(
			IN	:= FALSE,
		);
	END_IF
	bLastVisionConnected := TVision.bConnected;
END_IF
IF (TVision.bConnected) THEN (* check if vision software is still alive *)
	TAliveCheckTimer(
		IN	:= (bAliveCheck = TVision.bAlive),
		PT	:= t#10s,
	);
	bAliveCheck := TVision.bAlive;
	IF (TAliveCheckTimer.Q) THEN
		TVision.bConnected := FALSE;
	END_IF
END_IF
IF (TVision.bConnected) THEN
	CASE eVisionStep OF
		SP_RunStp0: (* Wait command *)
			TVision.bRequestDone := TRUE;
			IF (eVisionCommand <> VR_None) THEN
				TVision.eRequest := eVisionCommand;
				(*Write parameter here *)
				TVision.bRequestError := FALSE;
				TVision.bRequestDone := FALSE;
				eVisionStep := SP_RunStp1;
			END_IF
		SP_RunStp1: (* Wait command received by the vision*)
			IF (TVision.eRequest = VR_None) THEN
				eVisionStep := SP_RunStp0;
			END_IF
	END_CASE
ELSE
	(* No vision connected, reset interface and mark request error *)
	TVision.bRequestError := TRUE;
	TVision.bRequestDone := TRUE;
	TVision.bAlive := FALSE;
	TVision.bReady := FALSE;
	TVision.bSimRecipe := FALSE;
	TVision.eRequest := VR_None;
	TVision.acRefFileName := '';
	TVision.iUseModel := 0;
	TVision.iMaxModel := 0;
	TVision.TPartData.bPresent := FALSE;
	TVision.TPartData.bValid := FALSE;
	TVision.TPartData.lrScore := 0;
	TVision.TPartData.lrTheta := 0;
	TVision.TPartData.lrX := 0;
	TVision.TPartData.lrY := 0;
	eVisionStep := SP_RunStp0;
END_IF
eVisionCommand := VR_None;
bNotConnected := NOT TVision.bConnected;
bInSimulation := TVision.bSimRecipe;


IF NOT fbNtGetTime.Busy THEN
	bNtGetTime := NOT bNtGetTime;
END_IF

fbNtGetTime(
	START := 	bNtGetTime
);

IF NOT fbNtGetTime.Busy THEN
	TNow := fbNtGetTime.TIMESTR;
END_IF

IF bResetErrors THEN
	bNotReady := FALSE;
	bNotConnected := FALSE;
	sCurrentState.bInError := FALSE;
END_IF

IF bSimVision THEN
	IF bNotConnected OR bNotReady THEN
		sCurrentState.bInError := TRUE;
		IF (sCurrentState.eStatus <> MS_Manual) AND (sCurrentState.eStatus <> MS_Stopped) AND (sCurrentState.eStatus <> MS_Init) THEN
			sCurrentState.eStatus := MS_Ready;
		END_IF
	END_IF
	IF bNotConnected OR bNotReady OR bNewJob THEN
		sCurrentState.bInitDone := FALSE;
		IF (sCurrentState.eStatus <> MS_Manual) THEN
			sCurrentState.eStatus := MS_Stopped;
		END_IF
	END_IF
ELSE
	sCurrentState.bInitDone := TRUE;
	sCurrentState.bInError := FALSE;
END_IF

IF NOT bJobInProgress AND NOT bNotConnected THEN (* bypass when no recipe is loaded *)
	sCurrentState.bInitDone := TRUE;
	sCurrentState.bInError := FALSE;
	bNotConnected := FALSE;
	bNotReady := FALSE;
END_IF

sRunData.iMaxModel := TVision.iMaxModel;

sCurrentState.bWarning := bInSimulation;
bModuleError := sCurrentState.bInError;

sCurrentState.bRunning := (sCurrentState.eStatus = MS_Running);
IF (sCurrentState.eStatus <> MS_Running) THEN eRunStatus := RS_NotRunning; END_IF

END_FUNCTION_BLOCK

// ---- POUs/Handlers/UtilitiesHdl.TcPOU
FUNCTION_BLOCK UtilitiesHdl
(*
	Description 	: Bloc fonction de gestion des Utilities
	Auteur		: DRE
	Date		: 06.09.2016
	Version		: 1.00

	Modifications :

*)

VAR_INPUT
	bEnable						: BOOL;
	bDrivesAreOFF				: BOOL;
	b24VOK						: BOOL;
	b48VOK						: BOOL;
	bAirPressureOK				: BOOL;
	bVacuumPumpIsOn			: BOOL;
	bMainVacuumOK				: BOOL;
	bAspirationIsOn				: BOOL;
	bAspirationOK				: BOOL;
	bPowerOn					: BOOL;
	bResetErrors					: BOOL;
	bStopReq					: BOOL;
	bPauseReq					: BOOL;
	eCommand					: TModuleCommands;
	bTableAspiration13On			: BOOL;
	bTableAspiration24On			: BOOL;
	bLoaderBrushAspirationOn		: BOOL;
	bBrushAspirationOn			: BOOL;
	bSharpenAspirationOn			: BOOL;
	bLoaderVacuumInUse			: BOOL;
END_VAR
VAR_OUTPUT
	bModuleError					: BOOL;
	bVacuumPumpOn				: BOOL;
	bAspirationOn				: BOOL;
	bVacuumError				: BOOL;
	bAspirationError				: BOOL;
	bAirPressureError				: BOOL;
	b24VError					: BOOL;
	b48VError					: BOOL;
	bPowerError					: BOOL;
	bDrivePowerError				: BOOL;
	bTableAspiration13Vacuum		: BOOL;
	bTableAspiration13Blowing		: BOOL;
	bTableAspiration24Vacuum		: BOOL;
	bTableAspiration24Blowing		: BOOL;
	bLoaderBrushAspirationVacuum	: BOOL;
	bLoaderBrushAspirationBlowing	: BOOL;
	bBrushAspirationVacuum		: BOOL;
	bBrushAspirationBlowing		: BOOL;
	bSharpenAspirationVacuum	: BOOL;
	bSharpenAspirationBlowing		: BOOL;
	dwAspirationUseTime			: DWORD;
	dwVacuumUseTime			: DWORD;
END_VAR
VAR_IN_OUT
	sCurrentState					: TModuleData;
	TManualCmd					: TManUtilities;
END_VAR
VAR
	TPumpCheckTimer				: TON;
	TSupplyFilter				: TON;
	TVacuumOnTimer				: TON;
	TVacuumOffTimer				: TON;
	TVacuumOk					: TOF;
	TVacuumCounter				: RunningCounter;
	TAspirationCounter			: RunningCounter;

	TTableAspiration13			: FB_AspirationValve;
	TTableAspiration24			: FB_AspirationValve;
	TLoaderBrushAspiration		: FB_AspirationValve;
	TBrushAspiration				: FB_AspirationValve;
	TSharpenAspiration			: FB_AspirationValve;

	bLastLoaderVacuumUse		: BOOL;
	TShutdownVacuum				: TON;
	
	iDebug						: INT := 0;

END_VAR

IF (NOT sCurrentState.bStepMode) THEN
	sCurrentState.bWaitStep := FALSE;
END_IF

IF sCurrentState.eStatus<>MS_Stopped AND sCurrentState.eStatus<>MS_Ready THEN
	TVacuumOffTimer(IN := FALSE);
END_IF

TVacuumOk(IN := bMainVacuumOK, PT := t#5s);
TVacuumOnTimer(IN := bVacuumPumpOn, PT := t#10s);

CASE eCommand OF+
	MC_NoCmd :
		CASE sCurrentState.eStatus OF
			MS_Init :
				IF bEnable THEN
				CASE sCurrentState.eStep OF
					SP_InitStp1 : (* Start Pumps*)
						bVacuumPumpOn := TRUE;
						bAspirationOn := TRUE;
						TPumpCheckTimer(
							IN	:= FALSE
						);
						iDebug := 1;
						sCurrentState.eStep := SP_InitStp2;
					SP_InitStp2:
						TPumpCheckTimer(
							IN	:= TRUE,
							PT	:= t#20s,
						);
						IF bVacuumPumpIsOn AND bAspirationIsOn AND bAspirationOK THEN
							TPumpCheckTimer(
								IN	:= FALSE,
							);
							iDebug := 2;
							sCurrentState.eStep := SP_InitStp3;
						ELSIF TPumpCheckTimer.Q THEN
							IF NOT bVacuumPumpIsOn THEN 
								bVacuumError := TRUE; 
								iDebug := 3;
							END_IF
							IF NOT bAspirationIsOn THEN 
								bAspirationError := TRUE;
								iDebug := 4;
							END_IF
						END_IF
					SP_InitStp3:
						TPumpCheckTimer(
							IN	:= TRUE,
							PT	:= T#20S,
						);
						IF (bMainVacuumOK) THEN
							TPumpCheckTimer(
								IN	:= FALSE,
							);
							iDebug := 5;
							sCurrentState.eStep := SP_InitStp99;
						ELSIF TPumpCheckTimer.Q OR NOT bVacuumPumpIsOn THEN
							bVacuumError := TRUE;
							iDebug := 6;
						END_IF
						IF NOT bAspirationIsOn OR NOT bAspirationOK THEN
							bAspirationError := TRUE;
							iDebug := 7;
						END_IF
					SP_InitStp99 : (* Leave Init *)
						sCurrentState.eStep := SP_RunStp1;
						sCurrentState.eStatus := MS_Ready;
						sCurrentState.bInitDone := TRUE;
				END_CASE
				ELSE
					sCurrentState.eStatus := MS_Ready;
					sCurrentState.bInitDone := TRUE;
				END_IF
			MS_Running :
				IF bEnable AND  (NOT sCurrentState.bWaitStep) THEN
					CASE sCurrentState.eStep OF
						SP_RunStp1:
							IF bStopReq THEN
								sCurrentState.eStatus := MS_Ready;
							ELSIF bPauseReq THEN
								sCurrentState.eStatus := MS_Paused;
							ELSE
								bVacuumPumpOn := TRUE;
								bAspirationOn := TRUE;
								IF TVacuumOnTimer.Q THEN
									IF NOT bVacuumPumpIsOn OR NOT TVacuumOk.Q THEN
										bVacuumError := TRUE;
									END_IF
									IF NOT bAspirationIsOn OR NOT bAspirationOK THEN
										bAspirationError := TRUE;
									END_IF
								END_IF
							END_IF
					END_CASE
				END_IF
			MS_Manual :
				TManualCmd.b24VOK := b24VOK;
				TManualCmd.b48VOK := b48VOK;
				TManualCmd.bAirPressureOK := bAirPressureOK;
				TManualCmd.bDrivesIsOn := NOT bDrivesAreOFF;
				TManualCmd.bMainVacuumOK := bMainVacuumOK;
				TManualCmd.bAspirationOK := bAspirationOK;
				TManualCmd.bAspirationIsOn := bAspirationIsOn;
				TManualCmd.bPowerIsOn := bPowerOn;
				TManualCmd.TAspiration.Enable := TRUE;
				TManualCmd.TVacuum.Enable := TRUE;
				TManualCmd.TResetAspirationUseTime.Enable := TRUE;
				TManualCmd.TResetVacuumUseTime.Enable := TRUE;
				TManualCmd.dwAspirationUseTime := TAspirationCounter.dwHours;
				TManualCmd.dwVacuumUseTime := TVacuumCounter.dwHours;
				CASE sCurrentState.eStep OF
					SP_ManualStp0 :
						TManualCmd.TAspiration.Activate := bAspirationOn;
						TManualCmd.TVacuum.Activate := bVacuumPumpOn;
						TManualCmd.TResetAspirationUseTime.Activate := FALSE;
						TManualCmd.TResetVacuumUseTime.Activate := FALSE;
						sCurrentState.eStep := SP_ManualStp1;
					SP_ManualStp1:
						IF bStopReq THEN
							sCurrentState.eStatus := MS_Stopped;
						END_IF
						bAspirationOn := TManualCmd.TAspiration.Activate;
						bVacuumPumpOn := TManualCmd.TVacuum.Activate;
						IF (TManualCmd.TResetAspirationUseTime.Activate) THEN
							TAspirationCounter(bReset := TRUE);
							TManualCmd.TResetAspirationUseTime.Activate := FALSE;
						END_IF
						IF (TManualCmd.TResetVacuumUseTime.Activate) THEN
							TVacuumCounter(bReset := TRUE);
							TManualCmd.TResetVacuumUseTime.Activate := FALSE;
						END_IF
				END_CASE
		MS_Paused:
			IF bStopReq THEN
				sCurrentState.eStatus := MS_Ready;
			END_IF
		MS_Stopped:
			TVacuumOffTimer(IN:=bVacuumPumpOn AND NOT bLoaderVacuumInUse, PT := t#30s);
			IF TVacuumOffTimer.Q AND NOT bLoaderVacuumInUse THEN
				bVacuumPumpOn := FALSE;
				bAspirationOn := FALSE;
				sCurrentState.bInitDone := FALSE;
			END_IF
		END_CASE;
	MC_Init :
		sCurrentState.eStep := SP_InitStp1;
(*		IF sCurrentState.bInitDone THEN
			sCurrentState.eStep := SP_InitStp99;
		ELSE
			sCurrentState.eStep := SP_InitStp1;
		END_IF
*)		sCurrentState.eStatus := MS_Init;
	MC_Run :
		sCurrentState.eStatus := MS_Running;
	MC_Manual :
		sCurrentState.bInitDone := FALSE;
		sCurrentState.eStatus := MS_Manual;
		sCurrentState.eStep := SP_ManualStp0;
	MC_Stop :
		sCurrentState.eStatus := MS_Stopped;
END_CASE;

IF NOT bEnable THEN
	bModuleError	:= FALSE;
END_IF

TSupplyFilter(IN := NOT bResetErrors, PT := t#500ms);
IF TSupplyFilter.Q THEN
	IF NOT b24VOK 			THEN b24VError := TRUE; END_IF
	IF NOT b48VOK 			THEN b48VError := TRUE; END_IF
	IF bDrivesAreOFF 			THEN bDrivePowerError := TRUE; END_IF
	IF NOT bPowerOn 		THEN bPowerError := TRUE; END_IF
END_IF
IF NOT bAirPressureOK	 THEN bAirPressureError := TRUE; END_IF

TVacuumCounter(bStart := bVacuumPumpIsOn, bReset := FALSE);
TAspirationCounter(bStart := bAspirationIsOn, bReset := FALSE);
dwAspirationUseTime := TAspirationCounter.dwHours;
dwVacuumUseTime := TVacuumCounter.dwHours;


(*IF bAspirationOn OR bAspirationIsOn THEN*)
	(* Force at least 1 aspiration open *)
	bTableAspiration13On := bTableAspiration13On OR NOT (bTableAspiration24On OR bLoaderBrushAspirationOn OR bBrushAspirationOn OR bSharpenAspirationOn);
(*END_IF*)

TTableAspiration13(
	bEnableAspiration := bTableAspiration13On,
	bVacuumOn		=> bTableAspiration13Vacuum,
	bBlowOn			=> bTableAspiration13Blowing
);
TTableAspiration24(
	bEnableAspiration := bTableAspiration24On,
	bVacuumOn		=> bTableAspiration24Vacuum,
	bBlowOn			=> bTableAspiration24Blowing
);
TLoaderBrushAspiration(
	bEnableAspiration := bLoaderBrushAspirationOn,
	bVacuumOn		=> bLoaderBrushAspirationVacuum,
	bBlowOn			=> bLoaderBrushAspirationBlowing
);
TBrushAspiration(
	bEnableAspiration := bBrushAspirationOn,
	bVacuumOn		=> bBrushAspirationVacuum,
	bBlowOn			=> bBrushAspirationBlowing
);
TSharpenAspiration(
	bEnableAspiration := bSharpenAspirationOn,
	bVacuumOn		=> bSharpenAspirationVacuum,
	bBlowOn			=> bSharpenAspirationBlowing
);

IF bResetErrors THEN
	sCurrentState.bInError := FALSE;
	bVacuumError := FALSE;
	bAspirationError := FALSE;
	bAirPressureError := FALSE;
	b24VError := FALSE;
	b48VError := FALSE;
	bPowerError := FALSE;
	bDrivePowerError := FALSE;
END_IF

IF NOT bPowerOn OR bDrivesAreOFF OR NOT b24VOK OR NOT b48VOK OR NOT bAirPressureOK OR bVacuumError OR bAspirationError THEN
	sCurrentState.bInError := TRUE;
		IF (sCurrentState.eStatus <> MS_Manual) AND (sCurrentState.eStatus <> MS_Stopped) AND (sCurrentState.eStatus <> MS_Init) THEN
		sCurrentState.eStatus := MS_Ready;
	END_IF
END_IF

IF (NOT bPowerOn OR bVacuumError OR bAspirationError) THEN
	sCurrentState.bInitDone := FALSE;
	IF (sCurrentState.eStatus <> MS_Manual) THEN
		sCurrentState.eStatus := MS_Stopped;
	END_IF
END_IF


bModuleError := sCurrentState.bInError;

sCurrentState.bRunning := (sCurrentState.eStatus = MS_Running);

(* Force vacuum pump off if no vacuum on head for 1 hour *)
TShutdownVacuum(IN:=bVacuumPumpOn AND (bLoaderVacuumInUse = bLastLoaderVacuumUse), PT := t#60m);
bLastLoaderVacuumUse := bLoaderVacuumInUse;
IF TShutdownVacuum.Q THEN
	bVacuumPumpOn := FALSE;
	bAspirationOn := FALSE;
	sCurrentState.bInitDone := FALSE;
	sCurrentState.eStatus := MS_Stopped;
END_IF

END_FUNCTION_BLOCK

// ---- POUs/Controls/FB_AspirationValve.TcPOU
FUNCTION_BLOCK FB_AspirationValve
(*
	Description 	: Bloc fonction de gestion d'un module de mise sous vide
	Auteur		: DLA
	Date		: 26.03.2014
	Version		: 1.00

	Modifications :

*)
VAR_INPUT
	bEnableAspiration			: BOOL	:= FALSE;			(* Demande d'activation du vacuum *)
(*	tBlowingTime				: TIME	:= t#200ms;*)			(* Temps de soufflage à la coupure du vacuum *)
END_VAR
VAR_OUTPUT
	bVacuumOn				: BOOL	:= FALSE;			(* Activation du vacuum *)
	bBlowOn					: BOOL	:= FALSE;			(* Activation du soufflage *)
END_VAR
VAR
(*	TBlow					: TON;*)
END_VAR

(*La commande de vacuum est directement reliée à la requête*)
bVacuumOn := bEnableAspiration;
bBlowOn := NOT bEnableAspiration;

(*
(*On fait tourner les timers de détection de vacuum et de soufflage*)
TBlow(IN:=NOT bEnableAspiration,PT:=tBlowingTime);

IF bEnableAspiration THEN
	bBlowOn := FALSE;
ELSE
	(*On contrôle que le vacuum s'est bien coupé aprés le soufflage*)
	bBlowOn := NOT TBlow.Q;
END_IF
*)

END_FUNCTION_BLOCK

// ---- POUs/Controls/FB_CheckJack1_1.TcPOU
FUNCTION_BLOCK FB_CheckJack1_1
(*
	Description 	: Bloc fonction de gestion d'un module de mise sous vide
	Auteur		: DLA
	Date		: 26.03.2014
	Version		: 1.00

	Modifications :

*)
VAR_INPUT
	bJackGoOut	: BOOL;
	bJackIsOut	: BOOL;
	bResetErrors 	: BOOL;
	tTimeOut		: TIME			:= t#1s;
END_VAR
VAR_OUTPUT
	bJackError	: BOOL;
END_VAR
VAR
	T_Error		: TON;
	RSJackErr	: RS;
	bJackErr		: BOOL;
END_VAR

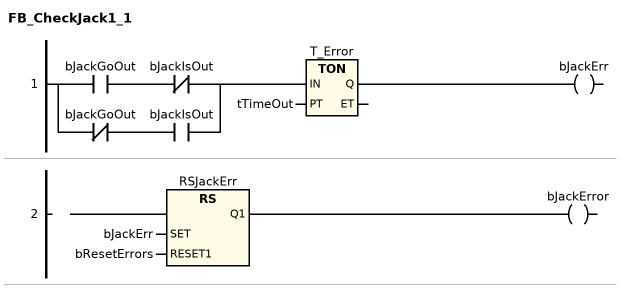
// NETWORK 1
T_Error(IN := bJackGoOut AND NOT bJackIsOut OR NOT bJackGoOut AND bJackIsOut, PT := tTimeOut); // TON
bJackErr := T_Error.Q;

// NETWORK 2
RSJackErr(SET := bJackErr, RESET1 := bResetErrors); // RS
bJackError := RSJackErr.Q1;

END_FUNCTION_BLOCK

// ---- POUs/utils/CalculatePosAngle.TcPOU
FUNCTION_BLOCK CalculatePosAngle
VAR_INPUT
	X1			: LREAL;
	X2			: LREAL;
	Y1			: LREAL;
	Y2			: LREAL;
END_VAR
VAR_OUTPUT
	alrResult		: ARRAY[0..2] OF LREAL;
END_VAR
VAR
END_VAR

alrResult[0] := X1;
alrResult[1] := Y1;
alrResult[2] := RAD_TO_DEG(ATAN((Y2-Y1)/(X2-X1)));

END_FUNCTION_BLOCK

// ---- POUs/utils/GetLoaderAxisFromTeachedAxis.TcPOU
FUNCTION GetLoaderAxisFromTeachedAxis : TLoaderAxis
VAR_INPUT
	eAxis	: TLoaderTeachedAxis;
END_VAR
VAR
END_VAR

CASE eAxis OF
	LTA_X:
		GetLoaderAxisFromTeachedAxis := LA_X;
	LTA_Y:
		GetLoaderAxisFromTeachedAxis := LA_Y;
	LTA_Z:
		GetLoaderAxisFromTeachedAxis := LA_Z1;
	LTA_THETA:
		GetLoaderAxisFromTeachedAxis := LA_THETA;
END_CASE

END_FUNCTION
